LIN {X 0,Y 443.866,Z 651.881,A -85,B 0,C 180,E1 8636.588,E2 8636.588} C_VEL
LIN {X 0,Y 424.776,Z 822.719,A -85,B 0,C 180,E1 8634.304,E2 8634.304} C_VEL
LIN {X 0,Y 420.494,Z 848.982,A -85,B 0,C 180,E1 8633.917,E2 8633.917} C_VEL
LIN {X 0,Y 414.112,Z 876.582,A -85,B 0,C 180,E1 8633.45,E2 8633.45} C_VEL
LIN {X 0,Y 407.99,Z 898.031,A -85,B 0,C 180,E1 8632.991,E2 8632.991} C_VEL
LIN {X 0,Y 400.93,Z 919.109,A -85,B 0,C 180,E1 8632.437,E2 8632.437} C_VEL
LIN {X 0,Y 392.51,Z 940.895,A -85,B 0,C 180,E1 8631.745,E2 8631.745} C_VEL
LIN {X 0,Y 380.405,Z 967.798,A -85,B 0,C 180,E1 8630.683,E2 8630.683} C_VEL
LIN {X 0,Y 369.913,Z 988.144,A -85,B 0,C 180,E1 8629.696,E2 8629.696} C_VEL
LIN {X 0,Y 359.109,Z 1007.066,A -85,B 0,C 180,E1 8628.598,E2 8628.598} C_VEL
LIN {X 0,Y 347.933,Z 1024.879,A -85,B 0,C 180,E1 8627.384,E2 8627.384} C_VEL
LIN {X 0,Y 333.364,Z 1046.114,A -85,B 0,C 180,E1 8625.643,E2 8625.643} C_VEL
LIN {X 0,Y 317.605,Z 1066.602,A -85,B 0,C 180,E1 8623.54,E2 8623.54} C_VEL
LIN {X 0,Y 304.112,Z 1082.781,A -85,B 0,C 180,E1 8621.51,E2 8621.51} C_VEL
LIN {X 0,Y 290.809,Z 1097.657,A -85,B 0,C 180,E1 8619.258,E2 8619.258} C_VEL
LIN {X 0,Y 275.048,Z 1114.162,A -85,B 0,C 180,E1 8616.201,E2 8616.201} C_VEL
LIN {X 0,Y 258.412,Z 1130.204,A -85,B 0,C 180,E1 8612.381,E2 8612.381} C_VEL
LIN {X 0,Y 245.42,Z 1142.096,A -85,B 0,C 180,E1 8608.821,E2 8608.821} C_VEL
LIN {X 0,Y 233.402,Z 1152.698,A -85,B 0,C 180,E1 8604.906,E2 8604.906} C_VEL
LIN {X 0,Y 221.406,Z 1163.045,A -85,B 0,C 180,E1 8600.148,E2 8600.148} C_VEL
LIN {X 0,Y 207.773,Z 1174.693,A -85,B 0,C 180,E1 8593.105,E2 8593.105} C_VEL
LIN {X 0,Y 199.178,Z 1182.245,A -85,B 0,C 180,E1 8587.041,E2 8587.041} C_VEL
LIN {X 0,Y 192.825,Z 1188.259,A -85,B 0,C 180,E1 8580.887,E2 8580.887} C_VEL
LIN {X 0,Y 188.308,Z 1193.142,A -85,B 0,C 180,E1 8574.466,E2 8574.466} C_VEL
LIN {X 0,Y 185.354,Z 1197.256,A -85,B 0,C 180,E1 8567.259,E2 8567.259} C_VEL
LIN {X 0,Y 184.079,Z 1200.28,A -85,B 0,C 180,E1 8559.378,E2 8559.378} C_VEL
LIN {X 0,Y 183.917,Z 1201.596,A -85,B 0,C 180,E1 8553.116,E2 8553.116} C_VEL
LIN {X 0,Y 183.913,Z 1201.997,A -85,B 0,C 180,E1 8547.507,E2 8547.507} C_VEL
LIN {X 0,Y 184.046,Z 1201.547,A -85,B 0,C 180,E1 8541.251,E2 8541.251} C_VEL
LIN {X 0,Y 185.236,Z 1199.666,A -85,B 0,C 180,E1 8533.377,E2 8533.377} C_VEL
LIN {X 0,Y 188.179,Z 1196.649,A -85,B 0,C 180,E1 8526.054,E2 8526.054} C_VEL
LIN {X 0,Y 192.95,Z 1192.697,A -85,B 0,C 180,E1 8519.343,E2 8519.343} C_VEL
LIN {X 0,Y 199.602,Z 1187.731,A -85,B 0,C 180,E1 8513.05,E2 8513.05} C_VEL
LIN {X 0,Y 208.813,Z 1181.234,A -85,B 0,C 180,E1 8506.786,E2 8506.786} C_VEL
LIN {X 0,Y 222.772,Z 1171.555,A -85,B 0,C 180,E1 8499.871,E2 8499.871} C_VEL
LIN {X 0,Y 236.844,Z 1161.509,A -85,B 0,C 180,E1 8494.593,E2 8494.593} C_VEL
LIN {X 0,Y 249.883,Z 1151.926,A -85,B 0,C 180,E1 8490.652,E2 8490.652} C_VEL
LIN {X 0,Y 263.952,Z 1141.12,A -85,B 0,C 180,E1 8487.104,E2 8487.104} C_VEL
LIN {X 0,Y 281.997,Z 1126.496,A -85,B 0,C 180,E1 8483.319,E2 8483.319} C_VEL
LIN {X 0,Y 300.287,Z 1110.217,A -85,B 0,C 180,E1 8480.122,E2 8480.122} C_VEL
LIN {X 0,Y 315.189,Z 1095.995,A -85,B 0,C 180,E1 8477.885,E2 8477.885} C_VEL
LIN {X 0,Y 329.674,Z 1081.143,A -85,B 0,C 180,E1 8475.968,E2 8475.968} C_VEL
LIN {X 0,Y 345.392,Z 1063.722,A -85,B 0,C 180,E1 8474.123,E2 8474.123} C_VEL
LIN {X 0,Y 363.236,Z 1041.735,A -85,B 0,C 180,E1 8472.263,E2 8472.263} C_VEL
LIN {X 0,Y 376.376,Z 1023.816,A -85,B 0,C 180,E1 8471.027,E2 8471.027} C_VEL
LIN {X 0,Y 388.341,Z 1005.955,A -85,B 0,C 180,E1 8469.997,E2 8469.997} C_VEL
LIN {X 0,Y 399.945,Z 986.891,A -85,B 0,C 180,E1 8469.072,E2 8469.072} C_VEL
LIN {X 0,Y 413.071,Z 962.812,A -85,B 0,C 180,E1 8468.109,E2 8468.109} C_VEL
LIN {X 0,Y 424.404,Z 938.434,A -85,B 0,C 180,E1 8467.327,E2 8467.327} C_VEL
LIN {X 0,Y 432.962,Z 917.372,A -85,B 0,C 180,E1 8466.777,E2 8466.777} C_VEL
LIN {X 0,Y 440.366,Z 896.336,A -85,B 0,C 180,E1 8466.323,E2 8466.323} C_VEL
LIN {X 0,Y 447.583,Z 872.049,A -85,B 0,C 180,E1 8465.902,E2 8465.902} C_VEL
LIN {X 0,Y 454.093,Z 843.665,A -85,B 0,C 180,E1 8465.507,E2 8465.507} C_VEL
LIN {X 0,Y 457.997,Z 820.681,A -85,B 0,C 180,E1 8465.208,E2 8465.208} C_VEL
LIN {X 0,Y 475.341,Z 679.715,A -85,B 0,C 180,E1 8463.437,E2 8463.437} C_VEL
LIN {X 0,Y 475.301,Z 680.039,A -85,B 0,C 180,E1 8463.377,E2 8463.377} C_VEL
LIN {X 0,Y 457.777,Z 822.091,A -85,B 0,C 180,E1 8461.612,E2 8461.612} C_VEL
LIN {X 0,Y 452.981,Z 849.333,A -85,B 0,C 180,E1 8461.256,E2 8461.256} C_VEL
LIN {X 0,Y 446.328,Z 876.186,A -85,B 0,C 180,E1 8460.853,E2 8460.853} C_VEL
LIN {X 0,Y 439.95,Z 897.255,A -85,B 0,C 180,E1 8460.454,E2 8460.454} C_VEL
LIN {X 0,Y 432.487,Z 918.241,A -85,B 0,C 180,E1 8459.972,E2 8459.972} C_VEL
LIN {X 0,Y 423.465,Z 940.191,A -85,B 0,C 180,E1 8459.362,E2 8459.362} C_VEL
LIN {X 0,Y 410.642,Z 966.852,A -85,B 0,C 180,E1 8458.444,E2 8458.444} C_VEL
LIN {X 0,Y 399.788,Z 986.536,A -85,B 0,C 180,E1 8457.615,E2 8457.615} C_VEL
LIN {X 0,Y 388.59,Z 1004.872,A -85,B 0,C 180,E1 8456.696,E2 8456.696} C_VEL
LIN {X 0,Y 376.533,Z 1022.797,A -85,B 0,C 180,E1 8455.644,E2 8455.644} C_VEL
LIN {X 0,Y 362.532,Z 1041.768,A -85,B 0,C 180,E1 8454.302,E2 8454.302} C_VEL
LIN {X 0,Y 344.561,Z 1063.586,A -85,B 0,C 180,E1 8452.39,E2 8452.39} C_VEL
LIN {X 0,Y 330.011,Z 1079.597,A -85,B 0,C 180,E1 8450.651,E2 8450.651} C_VEL
LIN {X 0,Y 315.549,Z 1094.316,A -85,B 0,C 180,E1 8448.721,E2 8448.721} C_VEL
LIN {X 0,Y 300.35,Z 1108.691,A -85,B 0,C 180,E1 8446.424,E2 8446.424} C_VEL
LIN {X 0,Y 281.29,Z 1125.37,A -85,B 0,C 180,E1 8443.053,E2 8443.053} C_VEL
LIN {X 0,Y 264.66,Z 1138.691,A -85,B 0,C 180,E1 8439.54,E2 8439.54} C_VEL
LIN {X 0,Y 250.503,Z 1149.41,A -85,B 0,C 180,E1 8435.975,E2 8435.975} C_VEL
LIN {X 0,Y 236.953,Z 1159.197,A -85,B 0,C 180,E1 8431.873,E2 8431.873} C_VEL
LIN {X 0,Y 221.703,Z 1169.857,A -85,B 0,C 180,E1 8426.08,E2 8426.08} C_VEL
LIN {X 0,Y 208.814,Z 1178.482,A -85,B 0,C 180,E1 8419.582,E2 8419.582} C_VEL
LIN {X 0,Y 199.873,Z 1184.582,A -85,B 0,C 180,E1 8413.499,E2 8413.499} C_VEL
LIN {X 0,Y 193.099,Z 1189.424,A -85,B 0,C 180,E1 8407.114,E2 8407.114} C_VEL
LIN {X 0,Y 187.925,Z 1193.548,A -85,B 0,C 180,E1 8399.657,E2 8399.657} C_VEL
LIN {X 0,Y 184.898,Z 1196.483,A -85,B 0,C 180,E1 8391.242,E2 8391.242} C_VEL
LIN {X 0,Y 184.057,Z 1197.676,A -85,B 0,C 180,E1 8384.471,E2 8384.471} C_VEL
LIN {X 0,Y 183.922,Z 1197.904,A -85,B 0,C 180,E1 8378.331,E2 8378.331} C_VEL
LIN {X 0,Y 183.937,Z 1197.343,A -85,B 0,C 180,E1 8372.492,E2 8372.492} C_VEL
LIN {X 0,Y 184.312,Z 1195.758,A -85,B 0,C 180,E1 8365.956,E2 8365.956} C_VEL
LIN {X 0,Y 185.733,Z 1193.043,A -85,B 0,C 180,E1 8359.14,E2 8359.14} C_VEL
LIN {X 0,Y 188.713,Z 1189.247,A -85,B 0,C 180,E1 8352.422,E2 8352.422} C_VEL
LIN {X 0,Y 193.222,Z 1184.592,A -85,B 0,C 180,E1 8346.195,E2 8346.195} C_VEL
LIN {X 0,Y 199.432,Z 1178.892,A -85,B 0,C 180,E1 8340.242,E2 8340.242} C_VEL
LIN {X 0,Y 207.741,Z 1171.761,A -85,B 0,C 180,E1 8334.383,E2 8334.383} C_VEL
LIN {X 0,Y 219.756,Z 1161.785,A -85,B 0,C 180,E1 8328.024,E2 8328.024} C_VEL
LIN {X 0,Y 233.341,Z 1150.204,A -85,B 0,C 180,E1 8322.523,E2 8322.523} C_VEL
LIN {X 0,Y 245.468,Z 1139.649,A -85,B 0,C 180,E1 8318.55,E2 8318.55} C_VEL
LIN {X 0,Y 258.583,Z 1127.787,A -85,B 0,C 180,E1 8314.942,E2 8314.942} C_VEL
LIN {X 0,Y 274.719,Z 1112.442,A -85,B 0,C 180,E1 8311.208,E2 8311.208} C_VEL
LIN {X 0,Y 291.052,Z 1095.466,A -85,B 0,C 180,E1 8308.009,E2 8308.009} C_VEL
LIN {X 0,Y 304.218,Z 1080.858,A -85,B 0,C 180,E1 8305.771,E2 8305.771} C_VEL
LIN {X 0,Y 317.272,Z 1065.327,A -85,B 0,C 180,E1 8303.791,E2 8303.791} C_VEL
LIN {X 0,Y 330.9,Z 1047.812,A -85,B 0,C 180,E1 8301.931,E2 8301.931} C_VEL
LIN {X 0,Y 346.823,Z 1025.164,A -85,B 0,C 180,E1 8299.978,E2 8299.978} C_VEL
LIN {X 0,Y 358.772,Z 1006.257,A -85,B 0,C 180,E1 8298.641,E2 8298.641} C_VEL
LIN {X 0,Y 369.602,Z 987.426,A -85,B 0,C 180,E1 8297.524,E2 8297.524} C_VEL
LIN {X 0,Y 379.674,Z 968.031,A -85,B 0,C 180,E1 8296.549,E2 8296.549} C_VEL
LIN {X 0,Y 391.196,Z 943.066,A -85,B 0,C 180,E1 8295.513,E2 8295.513} C_VEL
LIN {X 0,Y 400.78,Z 918.46,A -85,B 0,C 180,E1 8294.691,E2 8294.691} C_VEL
LIN {X 0,Y 407.769,Z 897.72,A -85,B 0,C 180,E1 8294.124,E2 8294.124} C_VEL
LIN {X 0,Y 413.868,Z 876.495,A -85,B 0,C 180,E1 8293.643,E2 8293.643} C_VEL
LIN {X 0,Y 419.539,Z 852.593,A -85,B 0,C 180,E1 8293.209,E2 8293.209} C_VEL
LIN {X 0,Y 424.62,Z 823.336,A -85,B 0,C 180,E1 8292.774,E2 8292.774} C_VEL
LIN {X 0,Y 432.472,Z 754.37,A -85,B 0,C 180,E1 8291.843,E2 8291.843} C_VEL
LIN {X 0,Y 443.846,Z 651.537,A -85,B 0,C 180,E1 8290.448,E2 8290.448} C_VEL
LIN {X 0,Y 442.904,Z 649.337,A -85,B 0,C 180,E1 8288.962,E2 8288.962} C_VEL
LIN {X 0,Y 441.948,Z 646.598,A -85,B 0,C 180,E1 8286.693,E2 8286.693} C_VEL
LIN {X 0,Y 441.415,Z 645.936,A -85,B 0,C 180,E1 8282.857,E2 8282.857} C_VEL
LIN {X 0,Y 441.662,Z 646.287,A -85,B 0,C 180,E1 8281.327,E2 8281.327} C_VEL
LIN {X 0,Y 441.718,Z 647.33,A -85,B 0,C 180,E1 8280.766,E2 8280.766} C_VEL
LIN {X 0,Y 441.574,Z 651.709,A -85,B 0,C 180,E1 8279.845,E2 8279.845} C_VEL
LIN {X 0,Y 441.535,Z 655.781,A -85,B 0,C 180,E1 8279.002,E2 8279.002} C_VEL
LIN {X 0,Y 441.696,Z 656.897,A -85,B 0,C 180,E1 8278.534,E2 8278.534} C_VEL
LIN {X 0,Y 442.275,Z 658.15,A -85,B 0,C 180,E1 8277.538,E2 8277.538} C_VEL
LIN {X 0,Y 423.591,Z 822.639,A -85,B 0,C 180,E1 8275.377,E2 8275.377} C_VEL
LIN {X 0,Y 419.223,Z 849.082,A -85,B 0,C 180,E1 8274.997,E2 8274.997} C_VEL
LIN {X 0,Y 412.777,Z 876.62,A -85,B 0,C 180,E1 8274.547,E2 8274.547} C_VEL
LIN {X 0,Y 406.591,Z 898.047,A -85,B 0,C 180,E1 8274.105,E2 8274.105} C_VEL
LIN {X 0,Y 399.454,Z 919.109,A -85,B 0,C 180,E1 8273.571,E2 8273.571} C_VEL
LIN {X 0,Y 390.939,Z 940.883,A -85,B 0,C 180,E1 8272.903,E2 8272.903} C_VEL
LIN {X 0,Y 378.497,Z 968.138,A -85,B 0,C 180,E1 8271.862,E2 8271.862} C_VEL
LIN {X 0,Y 367.593,Z 988.937,A -85,B 0,C 180,E1 8270.881,E2 8270.881} C_VEL
LIN {X 0,Y 356.811,Z 1007.503,A -85,B 0,C 180,E1 8269.831,E2 8269.831} C_VEL
LIN {X 0,Y 344.78,Z 1026.326,A -85,B 0,C 180,E1 8268.577,E2 8268.577} C_VEL
LIN {X 0,Y 328.296,Z 1049.535,A -85,B 0,C 180,E1 8266.672,E2 8266.672} C_VEL
LIN {X 0,Y 313.919,Z 1067.729,A -85,B 0,C 180,E1 8264.813,E2 8264.813} C_VEL
LIN {X 0,Y 300.669,Z 1083.249,A -85,B 0,C 180,E1 8262.893,E2 8262.893} C_VEL
LIN {X 0,Y 286.303,Z 1098.905,A -85,B 0,C 180,E1 8260.547,E2 8260.547} C_VEL
LIN {X 0,Y 268.106,Z 1117.205,A -85,B 0,C 180,E1 8257.094,E2 8257.094} C_VEL
LIN {X 0,Y 253.141,Z 1131.12,A -85,B 0,C 180,E1 8253.715,E2 8253.715} C_VEL
LIN {X 0,Y 239.782,Z 1142.917,A -85,B 0,C 180,E1 8250.15,E2 8250.15} C_VEL
LIN {X 0,Y 226.515,Z 1154.166,A -85,B 0,C 180,E1 8245.902,E2 8245.902} C_VEL
LIN {X 0,Y 211.151,Z 1166.776,A -85,B 0,C 180,E1 8239.674,E2 8239.674} C_VEL
LIN {X 0,Y 200.341,Z 1175.532,A -85,B 0,C 180,E1 8233.925,E2 8233.925} C_VEL
LIN {X 0,Y 191.817,Z 1182.641,A -85,B 0,C 180,E1 8227.958,E2 8227.958} C_VEL
LIN {X 0,Y 185.167,Z 1188.578,A -85,B 0,C 180,E1 8221.586,E2 8221.586} C_VEL
LIN {X 0,Y 180.081,Z 1193.81,A -85,B 0,C 180,E1 8214.259,E2 8214.259} C_VEL
LIN {X 0,Y 176.939,Z 1198.115,A -85,B 0,C 180,E1 8205.738,E2 8205.738} C_VEL
LIN {X 0,Y 176.03,Z 1200.441,A -85,B 0,C 180,E1 8198.492,E2 8198.492} C_VEL
LIN {X 0,Y 175.917,Z 1201.568,A -85,B 0,C 180,E1 8192.28,E2 8192.28} C_VEL
LIN {X 0,Y 175.914,Z 1201.879,A -85,B 0,C 180,E1 8186.415,E2 8186.415} C_VEL
LIN {X 0,Y 176.136,Z 1201.318,A -85,B 0,C 180,E1 8179.865,E2 8179.865} C_VEL
LIN {X 0,Y 177.612,Z 1199.394,A -85,B 0,C 180,E1 8171.964,E2 8171.964} C_VEL
LIN {X 0,Y 180.976,Z 1196.369,A -85,B 0,C 180,E1 8164.473,E2 8164.473} C_VEL
LIN {X 0,Y 186.011,Z 1192.573,A -85,B 0,C 180,E1 8157.849,E2 8157.849} C_VEL
LIN {X 0,Y 193.206,Z 1187.609,A -85,B 0,C 180,E1 8151.395,E2 8151.395} C_VEL
LIN {X 0,Y 202.782,Z 1181.279,A -85,B 0,C 180,E1 8145.163,E2 8145.163} C_VEL
LIN {X 0,Y 217.489,Z 1171.647,A -85,B 0,C 180,E1 8138.175,E2 8138.175} C_VEL
LIN {X 0,Y 232.357,Z 1161.509,A -85,B 0,C 180,E1 8132.834,E2 8132.834} C_VEL
LIN {X 0,Y 246.427,Z 1151.562,A -85,B 0,C 180,E1 8128.789,E2 8128.789} C_VEL
LIN {X 0,Y 262.191,Z 1139.838,A -85,B 0,C 180,E1 8125.044,E2 8125.044} C_VEL
LIN {X 0,Y 282.812,Z 1123.293,A -85,B 0,C 180,E1 8121.037,E2 8121.037} C_VEL
LIN {X 0,Y 298.379,Z 1109.731,A -85,B 0,C 180,E1 8118.5,E2 8118.5} C_VEL
LIN {X 0,Y 313.615,Z 1095.474,A -85,B 0,C 180,E1 8116.334,E2 8116.334} C_VEL
LIN {X 0,Y 329.267,Z 1079.67,A -85,B 0,C 180,E1 8114.378,E2 8114.378} C_VEL
LIN {X 0,Y 347.977,Z 1058.932,A -85,B 0,C 180,E1 8112.33,E2 8112.33} C_VEL
LIN {X 0,Y 363.426,Z 1039.824,A -85,B 0,C 180,E1 8110.834,E2 8110.834} C_VEL
LIN {X 0,Y 375.647,Z 1023.311,A -85,B 0,C 180,E1 8109.754,E2 8109.754} C_VEL
LIN {X 0,Y 388.023,Z 1005.022,A -85,B 0,C 180,E1 8108.745,E2 8108.745} C_VEL
LIN {X 0,Y 400.176,Z 985.189,A -85,B 0,C 180,E1 8107.832,E2 8107.832} C_VEL
LIN {X 0,Y 414.396,Z 958.757,A -85,B 0,C 180,E1 8106.848,E2 8106.848} C_VEL
LIN {X 0,Y 424.422,Z 937.2,A -85,B 0,C 180,E1 8106.201,E2 8106.201} C_VEL
LIN {X 0,Y 432.608,Z 917.166,A -85,B 0,C 180,E1 8105.704,E2 8105.704} C_VEL
LIN {X 0,Y 440.048,Z 896.191,A -85,B 0,C 180,E1 8105.272,E2 8105.272} C_VEL
LIN {X 0,Y 447.445,Z 871.471,A -85,B 0,C 180,E1 8104.864,E2 8104.864} C_VEL
LIN {X 0,Y 453.921,Z 843.316,A -85,B 0,C 180,E1 8104.489,E2 8104.489} C_VEL
LIN {X 0,Y 457.835,Z 820.461,A -85,B 0,C 180,E1 8104.2,E2 8104.2} C_VEL
LIN {X 0,Y 465.839,Z 756.902,A -85,B 0,C 180,E1 8103.416,E2 8103.416} C_VEL
LIN {X 0,Y 457.308,Z 824.05,A -85,B 0,C 180,E1 8102.593,E2 8102.593} C_VEL
LIN {X 0,Y 451.773,Z 853.513,A -85,B 0,C 180,E1 8102.217,E2 8102.217} C_VEL
LIN {X 0,Y 445.735,Z 877.298,A -85,B 0,C 180,E1 8101.868,E2 8101.868} C_VEL
LIN {X 0,Y 439.334,Z 898.118,A -85,B 0,C 180,E1 8101.487,E2 8101.487} C_VEL
LIN {X 0,Y 431.756,Z 919.132,A -85,B 0,C 180,E1 8101.022,E2 8101.022} C_VEL
LIN {X 0,Y 421.447,Z 943.771,A -85,B 0,C 180,E1 8100.355,E2 8100.355} C_VEL
LIN {X 0,Y 409.454,Z 967.959,A -85,B 0,C 180,E1 8099.539,E2 8099.539} C_VEL
LIN {X 0,Y 398.416,Z 987.662,A -85,B 0,C 180,E1 8098.737,E2 8098.737} C_VEL
LIN {X 0,Y 387.213,Z 1005.699,A -85,B 0,C 180,E1 8097.862,E2 8097.862} C_VEL
LIN {X 0,Y 374.286,Z 1024.573,A -85,B 0,C 180,E1 8096.784,E2 8096.784} C_VEL
LIN {X 0,Y 357.199,Z 1047.006,A -85,B 0,C 180,E1 8095.205,E2 8095.205} C_VEL
LIN {X 0,Y 341.112,Z 1065.81,A -85,B 0,C 180,E1 8093.547,E2 8093.547} C_VEL
LIN {X 0,Y 326.901,Z 1081.067,A -85,B 0,C 180,E1 8091.912,E2 8091.912} C_VEL
LIN {X 0,Y 312.319,Z 1095.543,A -85,B 0,C 180,E1 8090.045,E2 8090.045} C_VEL
LIN {X 0,Y 294.087,Z 1112.307,A -85,B 0,C 180,E1 8087.359,E2 8087.359} C_VEL
LIN {X 0,Y 275.458,Z 1127.784,A -85,B 0,C 180,E1 8084.132,E2 8084.132} C_VEL
LIN {X 0,Y 260.158,Z 1139.635,A -85,B 0,C 180,E1 8080.987,E2 8080.987} C_VEL
LIN {X 0,Y 245.71,Z 1150.175,A -85,B 0,C 180,E1 8077.476,E2 8077.476} C_VEL
LIN {X 0,Y 230.097,Z 1161.006,A -85,B 0,C 180,E1 8072.853,E2 8072.853} C_VEL
LIN {X 0,Y 213.993,Z 1171.545,A -85,B 0,C 180,E1 8066.757,E2 8066.757} C_VEL
LIN {X 0,Y 202.271,Z 1179.018,A -85,B 0,C 180,E1 8060.902,E2 8060.902} C_VEL
LIN {X 0,Y 193.019,Z 1184.94,A -85,B 0,C 180,E1 8054.788,E2 8054.788} C_VEL
LIN {X 0,Y 185.538,Z 1189.926,A -85,B 0,C 180,E1 8047.904,E2 8047.904} C_VEL
LIN {X 0,Y 179.5,Z 1194.401,A -85,B 0,C 180,E1 8038.987,E2 8038.987} C_VEL
LIN {X 0,Y 176.855,Z 1196.755,A -85,B 0,C 180,E1 8031.113,E2 8031.113} C_VEL
LIN {X 0,Y 176.057,Z 1197.796,A -85,B 0,C 180,E1 8024.471,E2 8024.471} C_VEL
LIN {X 0,Y 175.925,Z 1197.989,A -85,B 0,C 180,E1 8018.498,E2 8018.498} C_VEL
LIN {X 0,Y 175.935,Z 1197.468,A -85,B 0,C 180,E1 8012.606,E2 8012.606} C_VEL
LIN {X 0,Y 176.329,Z 1195.908,A -85,B 0,C 180,E1 8005.773,E2 8005.773} C_VEL
LIN {X 0,Y 177.957,Z 1193.062,A -85,B 0,C 180,E1 7998.331,E2 7998.331} C_VEL
LIN {X 0,Y 181.232,Z 1189.246,A -85,B 0,C 180,E1 7991.338,E2 7991.338} C_VEL
LIN {X 0,Y 186.119,Z 1184.571,A -85,B 0,C 180,E1 7984.887,E2 7984.887} C_VEL
LIN {X 0,Y 193.152,Z 1178.554,A -85,B 0,C 180,E1 7978.478,E2 7978.478} C_VEL
LIN {X 0,Y 202.972,Z 1170.664,A -85,B 0,C 180,E1 7971.993,E2 7971.993} C_VEL
LIN {X 0,Y 216.842,Z 1159.569,A -85,B 0,C 180,E1 7965.245,E2 7965.245} C_VEL
LIN {X 0,Y 229.431,Z 1149.313,A -85,B 0,C 180,E1 7960.494,E2 7960.494} C_VEL
LIN {X 0,Y 242.458,Z 1138.367,A -85,B 0,C 180,E1 7956.472,E2 7956.472} C_VEL
LIN {X 0,Y 258.969,Z 1123.858,A -85,B 0,C 180,E1 7952.271,E2 7952.271} C_VEL
LIN {X 0,Y 275.099,Z 1108.429,A -85,B 0,C 180,E1 7948.846,E2 7948.846} C_VEL
LIN {X 0,Y 288.91,Z 1094.347,A -85,B 0,C 180,E1 7946.319,E2 7946.319} C_VEL
LIN {X 0,Y 302.407,Z 1079.62,A -85,B 0,C 180,E1 7944.141,E2 7944.141} C_VEL
LIN {X 0,Y 317.118,Z 1062.327,A -85,B 0,C 180,E1 7942.034,E2 7942.034} C_VEL
LIN {X 0,Y 333.898,Z 1040.514,A -85,B 0,C 180,E1 7939.903,E2 7939.903} C_VEL
LIN {X 0,Y 346.756,Z 1022.021,A -85,B 0,C 180,E1 7938.44,E2 7938.44} C_VEL
LIN {X 0,Y 358.055,Z 1004.214,A -85,B 0,C 180,E1 7937.25,E2 7937.25} C_VEL
LIN {X 0,Y 369.494,Z 984.356,A -85,B 0,C 180,E1 7936.13,E2 7936.13} C_VEL
LIN {X 0,Y 382.413,Z 959.013,A -85,B 0,C 180,E1 7934.963,E2 7934.963} C_VEL
LIN {X 0,Y 392.303,Z 936.538,A -85,B 0,C 180,E1 7934.124,E2 7934.124} C_VEL
LIN {X 0,Y 400.001,Z 916.643,A -85,B 0,C 180,E1 7933.503,E2 7933.503} C_VEL
LIN {X 0,Y 407.058,Z 895.657,A -85,B 0,C 180,E1 7932.958,E2 7932.958} C_VEL
LIN {X 0,Y 413.773,Z 872.042,A -85,B 0,C 180,E1 7932.455,E2 7932.455} C_VEL
LIN {X 0,Y 420.13,Z 843.287,A -85,B 0,C 180,E1 7931.986,E2 7931.986} C_VEL
LIN {X 0,Y 423.868,Z 820.064,A -85,B 0,C 180,E1 7931.656,E2 7931.656} C_VEL
LIN {X 0,Y 442.263,Z 658.004,A -85,B 0,C 180,E1 7929.529,E2 7929.529} C_VEL
LIN {X 0,Y 440.949,Z 654.526,A -85,B 0,C 180,E1 7926.641,E2 7926.641} C_VEL
LIN {X 0,Y 440.437,Z 653.878,A -85,B 0,C 180,E1 7922.863,E2 7922.863} C_VEL
LIN {X 0,Y 441.06,Z 654.792,A -85,B 0,C 180,E1 7920.13,E2 7920.13} C_VEL
LIN {X 0,Y 441.696,Z 656.897,A -85,B 0,C 180,E1 7918.534,E2 7918.534} C_VEL
LIN {X 0,Y 441.712,Z 658.232,A -85,B 0,C 180,E1 7918.27,E2 7918.27} C_VEL
LIN {X 0,Y 441.466,Z 661.243,A -85,B 0,C 180,E1 7918.094,E2 7918.094} C_VEL
LIN {X 0,Y 440.865,Z 666.276,A -85,B 0,C 180,E1 7918.065,E2 7918.065} C_VEL
LIN {X 0,Y 439.256,Z 677.952,A -85,B 0,C 180,E1 7918.297,E2 7918.297} C_VEL
LIN {X 0,Y 438.927,Z 680.662,A -85,B 0,C 180,E1 7918.288,E2 7918.288} C_VEL
LIN {X 0,Y 422.55,Z 822.596,A -85,B 0,C 180,E1 7916.456,E2 7916.456} C_VEL
LIN {X 0,Y 418.103,Z 849.182,A -85,B 0,C 180,E1 7916.084,E2 7916.084} C_VEL
LIN {X 0,Y 411.594,Z 876.657,A -85,B 0,C 180,E1 7915.65,E2 7915.65} C_VEL
LIN {X 0,Y 405.347,Z 898.064,A -85,B 0,C 180,E1 7915.226,E2 7915.226} C_VEL
LIN {X 0,Y 398.309,Z 918.638,A -85,B 0,C 180,E1 7914.725,E2 7914.725} C_VEL
LIN {X 0,Y 390.004,Z 939.714,A -85,B 0,C 180,E1 7914.107,E2 7914.107} C_VEL
LIN {X 0,Y 378.143,Z 965.765,A -85,B 0,C 180,E1 7913.166,E2 7913.166} C_VEL
LIN {X 0,Y 366.369,Z 988.068,A -85,B 0,C 180,E1 7912.163,E2 7912.163} C_VEL
LIN {X 0,Y 355.715,Z 1006.254,A -85,B 0,C 180,E1 7911.179,E2 7911.179} C_VEL
LIN {X 0,Y 344.136,Z 1024.221,A -85,B 0,C 180,E1 7910.041,E2 7910.041} C_VEL
LIN {X 0,Y 330.058,Z 1044.154,A -85,B 0,C 180,E1 7908.518,E2 7908.518} C_VEL
LIN {X 0,Y 313.143,Z 1065.6,A -85,B 0,C 180,E1 7906.472,E2 7906.472} C_VEL
LIN {X 0,Y 298.811,Z 1082.158,A -85,B 0,C 180,E1 7904.51,E2 7904.51} C_VEL
LIN {X 0,Y 285.275,Z 1096.68,A -85,B 0,C 180,E1 7902.426,E2 7902.426} C_VEL
LIN {X 0,Y 270.948,Z 1111.019,A -85,B 0,C 180,E1 7899.928,E2 7899.928} C_VEL
LIN {X 0,Y 252.81,Z 1127.892,A -85,B 0,C 180,E1 7896.208,E2 7896.208} C_VEL
LIN {X 0,Y 237.104,Z 1141.381,A -85,B 0,C 180,E1 7892.32,E2 7892.32} C_VEL
LIN {X 0,Y 224.102,Z 1152.041,A -85,B 0,C 180,E1 7888.448,E2 7888.448} C_VEL
LIN {X 0,Y 211.554,Z 1161.968,A -85,B 0,C 180,E1 7883.919,E2 7883.919} C_VEL
LIN {X 0,Y 197.804,Z 1172.733,A -85,B 0,C 180,E1 7877.561,E2 7877.561} C_VEL
LIN {X 0,Y 186.342,Z 1181.575,A -85,B 0,C 180,E1 7870.363,E2 7870.363} C_VEL
LIN {X 0,Y 179.025,Z 1187.591,A -85,B 0,C 180,E1 7863.952,E2 7863.952} C_VEL
LIN {X 0,Y 173.59,Z 1192.569,A -85,B 0,C 180,E1 7857.067,E2 7857.067} C_VEL
LIN {X 0,Y 170.113,Z 1196.449,A -85,B 0,C 180,E1 7849.932,E2 7849.932} C_VEL
LIN {X 0,Y 168.431,Z 1199.141,A -85,B 0,C 180,E1 7843.037,E2 7843.037} C_VEL
LIN {X 0,Y 167.965,Z 1200.741,A -85,B 0,C 180,E1 7836.837,E2 7836.837} C_VEL
LIN {X 0,Y 167.921,Z 1201.538,A -85,B 0,C 180,E1 7831.365,E2 7831.365} C_VEL
LIN {X 0,Y 167.918,Z 1201.753,A -85,B 0,C 180,E1 7825.56,E2 7825.56} C_VEL
LIN {X 0,Y 168.243,Z 1201.119,A -85,B 0,C 180,E1 7818.69,E2 7818.69} C_VEL
LIN {X 0,Y 169.955,Z 1199.239,A -85,B 0,C 180,E1 7810.765,E2 7810.765} C_VEL
LIN {X 0,Y 173.609,Z 1196.309,A -85,B 0,C 180,E1 7803.217,E2 7803.217} C_VEL
LIN {X 0,Y 179.334,Z 1192.366,A -85,B 0,C 180,E1 7796.114,E2 7796.114} C_VEL
LIN {X 0,Y 187.335,Z 1187.269,A -85,B 0,C 180,E1 7789.372,E2 7789.372} C_VEL
LIN {X 0,Y 199.14,Z 1180.013,A -85,B 0,C 180,E1 7782.285,E2 7782.285} C_VEL
LIN {X 0,Y 214.822,Z 1170.137,A -85,B 0,C 180,E1 7775.461,E2 7775.461} C_VEL
LIN {X 0,Y 228.423,Z 1161.294,A -85,B 0,C 180,E1 7770.915,E2 7770.915} C_VEL
LIN {X 0,Y 242.511,Z 1151.711,A -85,B 0,C 180,E1 7767.057,E2 7767.057} C_VEL
LIN {X 0,Y 258.02,Z 1140.562,A -85,B 0,C 180,E1 7763.525,E2 7763.525} C_VEL
LIN {X 0,Y 277.477,Z 1125.604,A -85,B 0,C 180,E1 7759.868,E2 7759.868} C_VEL
LIN {X 0,Y 295.861,Z 1110.007,A -85,B 0,C 180,E1 7756.983,E2 7756.983} C_VEL
LIN {X 0,Y 311.399,Z 1095.784,A -85,B 0,C 180,E1 7754.88,E2 7754.88} C_VEL
LIN {X 0,Y 326.432,Z 1080.928,A -85,B 0,C 180,E1 7753.087,E2 7753.087} C_VEL
LIN {X 0,Y 343.592,Z 1062.503,A -85,B 0,C 180,E1 7751.283,E2 7751.283} C_VEL
LIN {X 0,Y 361.062,Z 1041.505,A -85,B 0,C 180,E1 7749.654,E2 7749.654} C_VEL
LIN {X 0,Y 374.579,Z 1023.563,A -85,B 0,C 180,E1 7748.519,E2 7748.519} C_VEL
LIN {X 0,Y 387.29,Z 1005.015,A -85,B 0,C 180,E1 7747.537,E2 7747.537} C_VEL
LIN {X 0,Y 399.64,Z 985.078,A -85,B 0,C 180,E1 7746.661,E2 7746.661} C_VEL
LIN {X 0,Y 414.002,Z 958.638,A -85,B 0,C 180,E1 7745.72,E2 7745.72} C_VEL
LIN {X 0,Y 424.129,Z 937.054,A -85,B 0,C 180,E1 7745.104,E2 7745.104} C_VEL
LIN {X 0,Y 432.35,Z 917.103,A -85,B 0,C 180,E1 7744.633,E2 7744.633} C_VEL
LIN {X 0,Y 439.636,Z 896.772,A -85,B 0,C 180,E1 7744.233,E2 7744.233} C_VEL
LIN {X 0,Y 446.579,Z 873.946,A -85,B 0,C 180,E1 7743.87,E2 7743.87} C_VEL
LIN {X 0,Y 453.649,Z 844.231,A -85,B 0,C 180,E1 7743.486,E2 7743.486} C_VEL
LIN {X 0,Y 454.632,Z 839.124,A -85,B 0,C 180,E1 7743.417,E2 7743.417} C_VEL
LIN {X 0,Y 449.814,Z 861.311,A -85,B 0,C 180,E1 7743.136,E2 7743.136} C_VEL
LIN {X 0,Y 443.17,Z 885.764,A -85,B 0,C 180,E1 7742.764,E2 7742.764} C_VEL
LIN {X 0,Y 433.816,Z 913.165,A -85,B 0,C 180,E1 7742.231,E2 7742.231} C_VEL
LIN {X 0,Y 425.128,Z 934.575,A -85,B 0,C 180,E1 7741.714,E2 7741.714} C_VEL
LIN {X 0,Y 416.022,Z 954.253,A -85,B 0,C 180,E1 7741.141,E2 7741.141} C_VEL
LIN {X 0,Y 405.585,Z 974.271,A -85,B 0,C 180,E1 7740.449,E2 7740.449} C_VEL
LIN {X 0,Y 391.461,Z 998.248,A -85,B 0,C 180,E1 7739.444,E2 7739.444} C_VEL
LIN {X 0,Y 376.954,Z 1019.723,A -85,B 0,C 180,E1 7738.328,E2 7738.328} C_VEL
LIN {X 0,Y 363.737,Z 1037.446,A -85,B 0,C 180,E1 7737.21,E2 7737.21} C_VEL
LIN {X 0,Y 350.31,Z 1053.905,A -85,B 0,C 180,E1 7735.982,E2 7735.982} C_VEL
LIN {X 0,Y 334.091,Z 1072.108,A -85,B 0,C 180,E1 7734.332,E2 7734.332} C_VEL
LIN {X 0,Y 314.931,Z 1091.418,A -85,B 0,C 180,E1 7732.117,E2 7732.117} C_VEL
LIN {X 0,Y 298.55,Z 1106.454,A -85,B 0,C 180,E1 7729.937,E2 7729.937} C_VEL
LIN {X 0,Y 283.52,Z 1119.24,A -85,B 0,C 180,E1 7727.65,E2 7727.65} C_VEL
LIN {X 0,Y 267.312,Z 1132.073,A -85,B 0,C 180,E1 7724.802,E2 7724.802} C_VEL
LIN {X 0,Y 247.117,Z 1146.823,A -85,B 0,C 180,E1 7720.517,E2 7720.517} C_VEL
LIN {X 0,Y 230.897,Z 1157.749,A -85,B 0,C 180,E1 7716.251,E2 7716.251} C_VEL
LIN {X 0,Y 217.546,Z 1166.301,A -85,B 0,C 180,E1 7711.938,E2 7711.938} C_VEL
LIN {X 0,Y 204.566,Z 1174.313,A -85,B 0,C 180,E1 7706.699,E2 7706.699} C_VEL
LIN {X 0,Y 190.491,Z 1182.827,A -85,B 0,C 180,E1 7699.098,E2 7699.098} C_VEL
LIN {X 0,Y 180.784,Z 1188.65,A -85,B 0,C 180,E1 7691.581,E2 7691.581} C_VEL
LIN {X 0,Y 174.626,Z 1192.588,A -85,B 0,C 180,E1 7684.53,E2 7684.53} C_VEL
LIN {X 0,Y 170.79,Z 1195.334,A -85,B 0,C 180,E1 7677.548,E2 7677.548} C_VEL
LIN {X 0,Y 168.733,Z 1197.106,A -85,B 0,C 180,E1 7670.562,E2 7670.562} C_VEL
LIN {X 0,Y 168.056,Z 1197.916,A -85,B 0,C 180,E1 7664.47,E2 7664.47} C_VEL
LIN {X 0,Y 167.925,Z 1198.067,A -85,B 0,C 180,E1 7658.561,E2 7658.561} C_VEL
LIN {X 0,Y 167.939,Z 1197.525,A -85,B 0,C 180,E1 7652.389,E2 7652.389} C_VEL
LIN {X 0,Y 168.348,Z 1196.057,A -85,B 0,C 180,E1 7645.572,E2 7645.572} C_VEL
LIN {X 0,Y 170.097,Z 1193.237,A -85,B 0,C 180,E1 7637.783,E2 7637.783} C_VEL
LIN {X 0,Y 173.611,Z 1189.447,A -85,B 0,C 180,E1 7630.486,E2 7630.486} C_VEL
LIN {X 0,Y 178.826,Z 1184.799,A -85,B 0,C 180,E1 7623.787,E2 7623.787} C_VEL
LIN {X 0,Y 185.904,Z 1179.104,A -85,B 0,C 180,E1 7617.464,E2 7617.464} C_VEL
LIN {X 0,Y 195.222,Z 1171.978,A -85,B 0,C 180,E1 7611.33,E2 7611.33} C_VEL
LIN {X 0,Y 208.516,Z 1162.01,A -85,B 0,C 180,E1 7604.792,E2 7604.792} C_VEL
LIN {X 0,Y 223.291,Z 1150.435,A -85,B 0,C 180,E1 7599.226,E2 7599.226} C_VEL
LIN {X 0,Y 236.357,Z 1139.882,A -85,B 0,C 180,E1 7595.27,E2 7595.27} C_VEL
LIN {X 0,Y 249.637,Z 1128.642,A -85,B 0,C 180,E1 7591.885,E2 7591.885} C_VEL
LIN {X 0,Y 265.159,Z 1114.737,A -85,B 0,C 180,E1 7588.527,E2 7588.527} C_VEL
LIN {X 0,Y 283.029,Z 1097.358,A -85,B 0,C 180,E1 7585.262,E2 7585.262} C_VEL
LIN {X 0,Y 298.027,Z 1081.484,A -85,B 0,C 180,E1 7582.904,E2 7582.904} C_VEL
LIN {X 0,Y 311.667,Z 1065.915,A -85,B 0,C 180,E1 7581.005,E2 7581.005} C_VEL
LIN {X 0,Y 325.246,Z 1049.136,A -85,B 0,C 180,E1 7579.307,E2 7579.307} C_VEL
LIN {X 0,Y 341.691,Z 1026.704,A -85,B 0,C 180,E1 7577.458,E2 7577.458} C_VEL
LIN {X 0,Y 354.884,Z 1006.48,A -85,B 0,C 180,E1 7576.109,E2 7576.109} C_VEL
LIN {X 0,Y 366.063,Z 987.564,A -85,B 0,C 180,E1 7575.055,E2 7575.055} C_VEL
LIN {X 0,Y 376.397,Z 968.181,A -85,B 0,C 180,E1 7574.146,E2 7574.146} C_VEL
LIN {X 0,Y 388.172,Z 943.287,A -85,B 0,C 180,E1 7573.182,E2 7573.182} C_VEL
LIN {X 0,Y 397.765,Z 919.288,A -85,B 0,C 180,E1 7572.434,E2 7572.434} C_VEL
LIN {X 0,Y 405.133,Z 897.942,A -85,B 0,C 180,E1 7571.889,E2 7571.889} C_VEL
LIN {X 0,Y 411.336,Z 876.829,A -85,B 0,C 180,E1 7571.443,E2 7571.443} C_VEL
LIN {X 0,Y 417.058,Z 853.258,A -85,B 0,C 180,E1 7571.044,E2 7571.044} C_VEL
LIN {X 0,Y 422.34,Z 823.715,A -85,B 0,C 180,E1 7570.628,E2 7570.628} C_VEL
LIN {X 0,Y 430.124,Z 757.619,A -85,B 0,C 180,E1 7569.769,E2 7569.769} C_VEL
LIN {X 0,Y 440.71,Z 664.924,A -85,B 0,C 180,E1 7568.579,E2 7568.579} C_VEL
LIN {X 0,Y 439.928,Z 662.433,A -85,B 0,C 180,E1 7566.525,E2 7566.525} C_VEL
LIN {X 0,Y 439.463,Z 661.831,A -85,B 0,C 180,E1 7562.806,E2 7562.806} C_VEL
LIN {X 0,Y 440.03,Z 662.673,A -85,B 0,C 180,E1 7560.26,E2 7560.26} C_VEL
LIN {X 0,Y 440.702,Z 665.212,A -85,B 0,C 180,E1 7558.484,E2 7558.484} C_VEL
LIN {X 0,Y 438.927,Z 680.662,A -85,B 0,C 180,E1 7558.288,E2 7558.288} C_VEL
LIN {X 0,Y 437.954,Z 688.363,A -85,B 0,C 180,E1 7558.319,E2 7558.319} C_VEL
LIN {X 0,Y 435.041,Z 708.976,A -85,B 0,C 180,E1 7558.879,E2 7558.879} C_VEL
LIN {X 0,Y 434.215,Z 715.583,A -85,B 0,C 180,E1 7558.895,E2 7558.895} C_VEL
LIN {X 0,Y 421.587,Z 823.061,A -85,B 0,C 180,E1 7557.532,E2 7557.532} C_VEL
LIN {X 0,Y 416.859,Z 850.668,A -85,B 0,C 180,E1 7557.156,E2 7557.156} C_VEL
LIN {X 0,Y 410.413,Z 877.247,A -85,B 0,C 180,E1 7556.75,E2 7556.75} C_VEL
LIN {X 0,Y 404.016,Z 898.837,A -85,B 0,C 180,E1 7556.338,E2 7556.338} C_VEL
LIN {X 0,Y 396.493,Z 920.426,A -85,B 0,C 180,E1 7555.828,E2 7555.828} C_VEL
LIN {X 0,Y 385.921,Z 946.393,A -85,B 0,C 180,E1 7555.071,E2 7555.071} C_VEL
LIN {X 0,Y 374.846,Z 969.443,A -85,B 0,C 180,E1 7554.228,E2 7554.228} C_VEL
LIN {X 0,Y 364.381,Z 988.862,A -85,B 0,C 180,E1 7553.374,E2 7553.374} C_VEL
LIN {X 0,Y 353.763,Z 1006.693,A -85,B 0,C 180,E1 7552.439,E2 7552.439} C_VEL
LIN {X 0,Y 341.399,Z 1025.54,A -85,B 0,C 180,E1 7551.278,E2 7551.278} C_VEL
LIN {X 0,Y 325.298,Z 1047.719,A -85,B 0,C 180,E1 7549.6,E2 7549.6} C_VEL
LIN {X 0,Y 309.497,Z 1067.101,A -85,B 0,C 180,E1 7547.755,E2 7547.755} C_VEL
LIN {X 0,Y 295.8,Z 1082.577,A -85,B 0,C 180,E1 7545.955,E2 7545.955} C_VEL
LIN {X 0,Y 281.99,Z 1097.054,A -85,B 0,C 180,E1 7543.922,E2 7543.922} C_VEL
LIN {X 0,Y 266.085,Z 1112.56,A -85,B 0,C 180,E1 7541.249,E2 7541.249} C_VEL
LIN {X 0,Y 246.894,Z 1129.69,A -85,B 0,C 180,E1 7537.419,E2 7537.419} C_VEL
LIN {X 0,Y 231.827,Z 1142.198,A -85,B 0,C 180,E1 7533.778,E2 7533.778} C_VEL
LIN {X 0,Y 218.428,Z 1152.765,A -85,B 0,C 180,E1 7529.899,E2 7529.899} C_VEL
LIN {X 0,Y 203.015,Z 1164.492,A -85,B 0,C 180,E1 7524.353,E2 7524.353} C_VEL
LIN {X 0,Y 189.071,Z 1174.663,A -85,B 0,C 180,E1 7517.761,E2 7517.761} C_VEL
LIN {X 0,Y 179.307,Z 1181.873,A -85,B 0,C 180,E1 7511.573,E2 7511.573} C_VEL
LIN {X 0,Y 171.507,Z 1187.908,A -85,B 0,C 180,E1 7504.842,E2 7504.842} C_VEL
LIN {X 0,Y 165.795,Z 1192.812,A -85,B 0,C 180,E1 7497.669,E2 7497.669} C_VEL
LIN {X 0,Y 161.908,Z 1196.944,A -85,B 0,C 180,E1 7489.48,E2 7489.48} C_VEL
LIN {X 0,Y 160.146,Z 1199.998,A -85,B 0,C 180,E1 7480.431,E2 7480.431} C_VEL
LIN {X 0,Y 159.918,Z 1201.302,A -85,B 0,C 180,E1 7473.585,E2 7473.585} C_VEL
LIN {X 0,Y 159.914,Z 1201.684,A -85,B 0,C 180,E1 7467.491,E2 7467.491} C_VEL
LIN {X 0,Y 160.078,Z 1201.359,A -85,B 0,C 180,E1 7460.654,E2 7460.654} C_VEL
LIN {X 0,Y 161.638,Z 1199.774,A -85,B 0,C 180,E1 7451.611,E2 7451.611} C_VEL
LIN {X 0,Y 166.031,Z 1196.453,A -85,B 0,C 180,E1 7442.286,E2 7442.286} C_VEL
LIN {X 0,Y 172.151,Z 1192.575,A -85,B 0,C 180,E1 7434.901,E2 7434.901} C_VEL
LIN {X 0,Y 180.635,Z 1187.546,A -85,B 0,C 180,E1 7427.951,E2 7427.951} C_VEL
LIN {X 0,Y 191.322,Z 1181.335,A -85,B 0,C 180,E1 7421.585,E2 7421.585} C_VEL
LIN {X 0,Y 206.904,Z 1172.238,A -85,B 0,C 180,E1 7414.763,E2 7414.763} C_VEL
LIN {X 0,Y 224.238,Z 1161.417,A -85,B 0,C 180,E1 7409.08,E2 7409.08} C_VEL
LIN {X 0,Y 238.827,Z 1151.861,A -85,B 0,C 180,E1 7405.272,E2 7405.272} C_VEL
LIN {X 0,Y 254.321,Z 1141.086,A -85,B 0,C 180,E1 7401.902,E2 7401.902} C_VEL
LIN {X 0,Y 273.091,Z 1127.124,A -85,B 0,C 180,E1 7398.511,E2 7398.511} C_VEL
LIN {X 0,Y 292.685,Z 1111.041,A -85,B 0,C 180,E1 7395.559,E2 7395.559} C_VEL
LIN {X 0,Y 308.742,Z 1096.698,A -85,B 0,C 180,E1 7393.484,E2 7393.484} C_VEL
LIN {X 0,Y 323.949,Z 1082.001,A -85,B 0,C 180,E1 7391.754,E2 7391.754} C_VEL
LIN {X 0,Y 339.318,Z 1065.884,A -85,B 0,C 180,E1 7390.204,E2 7390.204} C_VEL
LIN {X 0,Y 356.983,Z 1045.586,A -85,B 0,C 180,E1 7388.622,E2 7388.622} C_VEL
LIN {X 0,Y 372.994,Z 1024.771,A -85,B 0,C 180,E1 7387.33,E2 7387.33} C_VEL
LIN {X 0,Y 385.64,Z 1006.652,A -85,B 0,C 180,E1 7386.401,E2 7386.401} C_VEL
LIN {X 0,Y 397.297,Z 988.232,A -85,B 0,C 180,E1 7385.613,E2 7385.613} C_VEL
LIN {X 0,Y 408.44,Z 968.683,A -85,B 0,C 180,E1 7384.911,E2 7384.911} C_VEL
LIN {X 0,Y 421.056,Z 943.596,A -85,B 0,C 180,E1 7384.174,E2 7384.174} C_VEL
LIN {X 0,Y 431.294,Z 919.487,A -85,B 0,C 180,E1 7383.611,E2 7383.611} C_VEL
LIN {X 0,Y 435.489,Z 908.683,A -85,B 0,C 180,E1 7383.394,E2 7383.394} C_VEL
LIN {X 0,Y 425.459,Z 933.511,A -85,B 0,C 180,E1 7382.834,E2 7382.834} C_VEL
LIN {X 0,Y 416.272,Z 953.314,A -85,B 0,C 180,E1 7382.291,E2 7382.291} C_VEL
LIN {X 0,Y 406.111,Z 972.757,A -85,B 0,C 180,E1 7381.657,E2 7381.657} C_VEL
LIN {X 0,Y 393.986,Z 993.459,A -85,B 0,C 180,E1 7380.853,E2 7380.853} C_VEL
LIN {X 0,Y 377.452,Z 1018.232,A -85,B 0,C 180,E1 7379.66,E2 7379.66} C_VEL
LIN {X 0,Y 363.836,Z 1036.383,A -85,B 0,C 180,E1 7378.583,E2 7378.583} C_VEL
LIN {X 0,Y 349.837,Z 1053.384,A -85,B 0,C 180,E1 7377.379,E2 7377.379} C_VEL
LIN {X 0,Y 334.79,Z 1070.099,A -85,B 0,C 180,E1 7375.943,E2 7375.943} C_VEL
LIN {X 0,Y 315.748,Z 1089.321,A -85,B 0,C 180,E1 7373.89,E2 7373.89} C_VEL
LIN {X 0,Y 298.079,Z 1105.339,A -85,B 0,C 180,E1 7371.701,E2 7371.701} C_VEL
LIN {X 0,Y 282.682,Z 1118.234,A -85,B 0,C 180,E1 7369.512,E2 7369.512} C_VEL
LIN {X 0,Y 266.877,Z 1130.518,A -85,B 0,C 180,E1 7366.929,E2 7366.929} C_VEL
LIN {X 0,Y 250.033,Z 1142.698,A -85,B 0,C 180,E1 7363.686,E2 7363.686} C_VEL
LIN {X 0,Y 229.447,Z 1156.384,A -85,B 0,C 180,E1 7358.795,E2 7358.795} C_VEL
LIN {X 0,Y 214.249,Z 1165.752,A -85,B 0,C 180,E1 7354.249,E2 7354.249} C_VEL
LIN {X 0,Y 201.116,Z 1173.487,A -85,B 0,C 180,E1 7349.325,E2 7349.325} C_VEL
LIN {X 0,Y 189.006,Z 1180.397,A -85,B 0,C 180,E1 7343.523,E2 7343.523} C_VEL
LIN {X 0,Y 176.76,Z 1187.376,A -85,B 0,C 180,E1 7335.457,E2 7335.457} C_VEL
LIN {X 0,Y 168.164,Z 1192.27,A -85,B 0,C 180,E1 7326.907,E2 7326.907} C_VEL
LIN {X 0,Y 163.465,Z 1195.249,A -85,B 0,C 180,E1 7319.297,E2 7319.297} C_VEL
LIN {X 0,Y 160.982,Z 1197.11,A -85,B 0,C 180,E1 7311.88,E2 7311.88} C_VEL
LIN {X 0,Y 160.103,Z 1197.993,A -85,B 0,C 180,E1 7305.206,E2 7305.206} C_VEL
LIN {X 0,Y 159.925,Z 1198.144,A -85,B 0,C 180,E1 7298.63,E2 7298.63} C_VEL
LIN {X 0,Y 159.937,Z 1197.65,A -85,B 0,C 180,E1 7292.508,E2 7292.508} C_VEL
LIN {X 0,Y 160.369,Z 1196.206,A -85,B 0,C 180,E1 7285.351,E2 7285.351} C_VEL
LIN {X 0,Y 162.381,Z 1193.255,A -85,B 0,C 180,E1 7276.831,E2 7276.831} C_VEL
LIN {X 0,Y 166.256,Z 1189.445,A -85,B 0,C 180,E1 7269.217,E2 7269.217} C_VEL
LIN {X 0,Y 171.92,Z 1184.776,A -85,B 0,C 180,E1 7262.273,E2 7262.273} C_VEL
LIN {X 0,Y 179.939,Z 1178.764,A -85,B 0,C 180,E1 7255.474,E2 7255.474} C_VEL
LIN {X 0,Y 191.439,Z 1170.533,A -85,B 0,C 180,E1 7248.448,E2 7248.448} C_VEL
LIN {X 0,Y 206.376,Z 1159.658,A -85,B 0,C 180,E1 7241.746,E2 7241.746} C_VEL
LIN {X 0,Y 219.546,Z 1149.792,A -85,B 0,C 180,E1 7237.157,E2 7237.157} C_VEL
LIN {X 0,Y 233.167,Z 1139.155,A -85,B 0,C 180,E1 7233.26,E2 7233.26} C_VEL
LIN {X 0,Y 248.424,Z 1126.585,A -85,B 0,C 180,E1 7229.616,E2 7229.616} C_VEL
LIN {X 0,Y 267.669,Z 1109.415,A -85,B 0,C 180,E1 7225.811,E2 7225.811} C_VEL
LIN {X 0,Y 282.122,Z 1095.405,A -85,B 0,C 180,E1 7223.378,E2 7223.378} C_VEL
LIN {X 0,Y 296.18,Z 1080.759,A -85,B 0,C 180,E1 7221.294,E2 7221.294} C_VEL
LIN {X 0,Y 310.582,Z 1064.541,A -85,B 0,C 180,E1 7219.395,E2 7219.395} C_VEL
LIN {X 0,Y 327.042,Z 1044.309,A -85,B 0,C 180,E1 7217.471,E2 7217.471} C_VEL
LIN {X 0,Y 342.035,Z 1023.544,A -85,B 0,C 180,E1 7215.898,E2 7215.898} C_VEL
LIN {X 0,Y 353.654,Z 1005.868,A -85,B 0,C 180,E1 7214.782,E2 7214.782} C_VEL
LIN {X 0,Y 364.893,Z 987.035,A -85,B 0,C 180,E1 7213.775,E2 7213.775} C_VEL
LIN {X 0,Y 375.877,Z 966.588,A -85,B 0,C 180,E1 7212.861,E2 7212.861} C_VEL
LIN {X 0,Y 388.471,Z 939.631,A -85,B 0,C 180,E1 7211.883,E2 7211.883} C_VEL
LIN {X 0,Y 397.074,Z 918.12,A -85,B 0,C 180,E1 7211.251,E2 7211.251} C_VEL
LIN {X 0,Y 404.281,Z 897.329,A -85,B 0,C 180,E1 7210.745,E2 7210.745} C_VEL
LIN {X 0,Y 410.605,Z 875.881,A -85,B 0,C 180,E1 7210.313,E2 7210.313} C_VEL
LIN {X 0,Y 417.073,Z 849.06,A -85,B 0,C 180,E1 7209.888,E2 7209.888} C_VEL
LIN {X 0,Y 421.696,Z 821.911,A -85,B 0,C 180,E1 7209.521,E2 7209.521} C_VEL
LIN {X 0,Y 437.077,Z 690.752,A -85,B 0,C 180,E1 7207.862,E2 7207.862} C_VEL
LIN {X 0,Y 439.289,Z 671.765,A -85,B 0,C 180,E1 7207.625,E2 7207.625} C_VEL
LIN {X 0,Y 438.909,Z 670.34,A -85,B 0,C 180,E1 7206.409,E2 7206.409} C_VEL
LIN {X 0,Y 438.482,Z 669.763,A -85,B 0,C 180,E1 7202.859,E2 7202.859} C_VEL
LIN {X 0,Y 439.003,Z 670.553,A -85,B 0,C 180,E1 7200.392,E2 7200.392} C_VEL
LIN {X 0,Y 439.269,Z 672.096,A -85,B 0,C 180,E1 7199.44,E2 7199.44} C_VEL
LIN {X 0,Y 434.215,Z 715.583,A -85,B 0,C 180,E1 7198.895,E2 7198.895} C_VEL
LIN {X 0,Y 433.243,Z 723.285,A -85,B 0,C 180,E1 7198.93,E2 7198.93} C_VEL
LIN {X 0,Y 430.374,Z 743.893,A -85,B 0,C 180,E1 7199.506,E2 7199.506} C_VEL
LIN {X 0,Y 429.55,Z 750.5,A -85,B 0,C 180,E1 7199.523,E2 7199.523} C_VEL
LIN {X 0,Y 420.683,Z 824.092,A -85,B 0,C 180,E1 7198.606,E2 7198.606} C_VEL
LIN {X 0,Y 415.534,Z 852.854,A -85,B 0,C 180,E1 7198.224,E2 7198.224} C_VEL
LIN {X 0,Y 409.414,Z 877.695,A -85,B 0,C 180,E1 7197.858,E2 7197.858} C_VEL
LIN {X 0,Y 403.083,Z 898.839,A -85,B 0,C 180,E1 7197.471,E2 7197.471} C_VEL
LIN {X 0,Y 395.49,Z 920.424,A -85,B 0,C 180,E1 7196.984,E2 7196.984} C_VEL
LIN {X 0,Y 385.078,Z 945.814,A -85,B 0,C 180,E1 7196.278,E2 7196.278} C_VEL
LIN {X 0,Y 373.728,Z 969.208,A -85,B 0,C 180,E1 7195.462,E2 7195.462} C_VEL
LIN {X 0,Y 362.907,Z 989.05,A -85,B 0,C 180,E1 7194.625,E2 7194.625} C_VEL
LIN {X 0,Y 352.062,Z 1007.006,A -85,B 0,C 180,E1 7193.719,E2 7193.719} C_VEL
LIN {X 0,Y 339.292,Z 1026.175,A -85,B 0,C 180,E1 7192.579,E2 7192.579} C_VEL
LIN {X 0,Y 322.039,Z 1049.368,A -85,B 0,C 180,E1 7190.864,E2 7190.864} C_VEL
LIN {X 0,Y 306.917,Z 1067.558,A -85,B 0,C 180,E1 7189.175,E2 7189.175} C_VEL
LIN {X 0,Y 292.465,Z 1083.538,A -85,B 0,C 180,E1 7187.361,E2 7187.361} C_VEL
LIN {X 0,Y 276.842,Z 1099.487,A -85,B 0,C 180,E1 7185.141,E2 7185.141} C_VEL
LIN {X 0,Y 257.181,Z 1117.763,A -85,B 0,C 180,E1 7181.879,E2 7181.879} C_VEL
LIN {X 0,Y 241.38,Z 1131.252,A -85,B 0,C 180,E1 7178.749,E2 7178.749} C_VEL
LIN {X 0,Y 226.707,Z 1143.013,A -85,B 0,C 180,E1 7175.303,E2 7175.303} C_VEL
LIN {X 0,Y 210.696,Z 1155.161,A -85,B 0,C 180,E1 7170.738,E2 7170.738} C_VEL
LIN {X 0,Y 193.868,Z 1167.189,A -85,B 0,C 180,E1 7164.574,E2 7164.574} C_VEL
LIN {X 0,Y 181.908,Z 1175.498,A -85,B 0,C 180,E1 7158.853,E2 7158.853} C_VEL
LIN {X 0,Y 171.787,Z 1182.578,A -85,B 0,C 180,E1 7152.466,E2 7152.466} C_VEL
LIN {X 0,Y 163.36,Z 1188.747,A -85,B 0,C 180,E1 7145.123,E2 7145.123} C_VEL
LIN {X 0,Y 156.297,Z 1194.652,A -85,B 0,C 180,E1 7135.379,E2 7135.379} C_VEL
LIN {X 0,Y 153.086,Z 1198.166,A -85,B 0,C 180,E1 7126.701,E2 7126.701} C_VEL
LIN {X 0,Y 152.057,Z 1200.229,A -85,B 0,C 180,E1 7119.08,E2 7119.08} C_VEL
LIN {X 0,Y 151.917,Z 1201.299,A -85,B 0,C 180,E1 7112.263,E2 7112.263} C_VEL
LIN {X 0,Y 151.916,Z 1201.644,A -85,B 0,C 180,E1 7105.848,E2 7105.848} C_VEL
LIN {X 0,Y 152.278,Z 1201.139,A -85,B 0,C 180,E1 7098.256,E2 7098.256} C_VEL
LIN {X 0,Y 154.596,Z 1199.125,A -85,B 0,C 180,E1 7088.649,E2 7088.649} C_VEL
LIN {X 0,Y 159.204,Z 1196.149,A -85,B 0,C 180,E1 7080.255,E2 7080.255} C_VEL
LIN {X 0,Y 166.145,Z 1192.163,A -85,B 0,C 180,E1 7072.568,E2 7072.568} C_VEL
LIN {X 0,Y 175.673,Z 1186.945,A -85,B 0,C 180,E1 7065.355,E2 7065.355} C_VEL
LIN {X 0,Y 189.816,Z 1179.308,A -85,B 0,C 180,E1 7057.803,E2 7057.803} C_VEL
LIN {X 0,Y 206.902,Z 1169.528,A -85,B 0,C 180,E1 7051.201,E2 7051.201} C_VEL
LIN {X 0,Y 221.757,Z 1160.633,A -85,B 0,C 180,E1 7046.781,E2 7046.781} C_VEL
LIN {X 0,Y 236.942,Z 1150.996,A -85,B 0,C 180,E1 7043.085,E2 7043.085} C_VEL
LIN {X 0,Y 253.794,Z 1139.572,A -85,B 0,C 180,E1 7039.683,E2 7039.683} C_VEL
LIN {X 0,Y 275.717,Z 1123.331,A -85,B 0,C 180,E1 7036.056,E2 7036.056} C_VEL
LIN {X 0,Y 293.234,Z 1109.041,A -85,B 0,C 180,E1 7033.645,E2 7033.645} C_VEL
LIN {X 0,Y 308.928,Z 1095.172,A -85,B 0,C 180,E1 7031.766,E2 7031.766} C_VEL
LIN {X 0,Y 324.96,Z 1079.806,A -85,B 0,C 180,E1 7030.07,E2 7030.07} C_VEL
LIN {X 0,Y 344.272,Z 1059.456,A -85,B 0,C 180,E1 7028.284,E2 7028.284} C_VEL
LIN {X 0,Y 360.595,Z 1040.112,A -85,B 0,C 180,E1 7026.946,E2 7026.946} C_VEL
LIN {X 0,Y 373.968,Z 1022.701,A -85,B 0,C 180,E1 7025.961,E2 7025.961} C_VEL
LIN {X 0,Y 386.476,Z 1004.801,A -85,B 0,C 180,E1 7025.102,E2 7025.102} C_VEL
LIN {X 0,Y 399.077,Z 984.846,A -85,B 0,C 180,E1 7024.311,E2 7024.311} C_VEL
LIN {X 0,Y 413.696,Z 958.399,A -85,B 0,C 180,E1 7023.463,E2 7023.463} C_VEL
LIN {X 0,Y 415.307,Z 955.152,A -85,B 0,C 180,E1 7023.359,E2 7023.359} C_VEL
LIN {X 0,Y 404.118,Z 976.118,A -85,B 0,C 180,E1 7022.695,E2 7022.695} C_VEL
LIN {X 0,Y 388.617,Z 1001.435,A -85,B 0,C 180,E1 7021.71,E2 7021.71} C_VEL
LIN {X 0,Y 374.97,Z 1021.068,A -85,B 0,C 180,E1 7020.764,E2 7020.764} C_VEL
LIN {X 0,Y 361.95,Z 1038.06,A -85,B 0,C 180,E1 7019.781,E2 7019.781} C_VEL
LIN {X 0,Y 347.553,Z 1055.198,A -85,B 0,C 180,E1 7018.603,E2 7018.603} C_VEL
LIN {X 0,Y 329.423,Z 1074.816,A -85,B 0,C 180,E1 7016.938,E2 7016.938} C_VEL
LIN {X 0,Y 311.022,Z 1092.511,A -85,B 0,C 180,E1 7015.02,E2 7015.02} C_VEL
LIN {X 0,Y 295.084,Z 1106.591,A -85,B 0,C 180,E1 7013.118,E2 7013.118} C_VEL
LIN {X 0,Y 278.974,Z 1119.722,A -85,B 0,C 180,E1 7010.926,E2 7010.926} C_VEL
LIN {X 0,Y 260.645,Z 1133.513,A -85,B 0,C 180,E1 7008.015,E2 7008.015} C_VEL
LIN {X 0,Y 240.042,Z 1147.58,A -85,B 0,C 180,E1 7004.043,E2 7004.043} C_VEL
LIN {X 0,Y 223.346,Z 1158.066,A -85,B 0,C 180,E1 7000.07,E2 7000.07} C_VEL
LIN {X 0,Y 208.429,Z 1166.856,A -85,B 0,C 180,E1 6995.707,E2 6995.707} C_VEL
LIN {X 0,Y 193.571,Z 1175.177,A -85,B 0,C 180,E1 6990.201,E2 6990.201} C_VEL
LIN {X 0,Y 177.454,Z 1183.756,A -85,B 0,C 180,E1 6982.076,E2 6982.076} C_VEL
LIN {X 0,Y 167.394,Z 1189.019,A -85,B 0,C 180,E1 6974.815,E2 6974.815} C_VEL
LIN {X 0,Y 160.168,Z 1192.913,A -85,B 0,C 180,E1 6967.267,E2 6967.267} C_VEL
LIN {X 0,Y 155.363,Z 1195.73,A -85,B 0,C 180,E1 6959.282,E2 6959.282} C_VEL
LIN {X 0,Y 152.879,Z 1197.431,A -85,B 0,C 180,E1 6951.485,E2 6951.485} C_VEL
LIN {X 0,Y 152.054,Z 1198.156,A -85,B 0,C 180,E1 6944.47,E2 6944.47} C_VEL
LIN {X 0,Y 151.922,Z 1198.197,A -85,B 0,C 180,E1 6938.325,E2 6938.325} C_VEL
LIN {X 0,Y 151.948,Z 1197.638,A -85,B 0,C 180,E1 6931.886,E2 6931.886} C_VEL
LIN {X 0,Y 152.487,Z 1196.132,A -85,B 0,C 180,E1 6924.356,E2 6924.356} C_VEL
LIN {X 0,Y 154.712,Z 1193.272,A -85,B 0,C 180,E1 6915.784,E2 6915.784} C_VEL
LIN {X 0,Y 158.99,Z 1189.443,A -85,B 0,C 180,E1 6907.832,E2 6907.832} C_VEL
LIN {X 0,Y 165.141,Z 1184.753,A -85,B 0,C 180,E1 6900.632,E2 6900.632} C_VEL
LIN {X 0,Y 173.651,Z 1178.788,A -85,B 0,C 180,E1 6893.72,E2 6893.72} C_VEL
LIN {X 0,Y 185.975,Z 1170.466,A -85,B 0,C 180,E1 6886.515,E2 6886.515} C_VEL
LIN {X 0,Y 201.052,Z 1159.991,A -85,B 0,C 180,E1 6880.016,E2 6880.016} C_VEL
LIN {X 0,Y 214.735,Z 1150.154,A -85,B 0,C 180,E1 6875.429,E2 6875.429} C_VEL
LIN {X 0,Y 228.814,Z 1139.547,A -85,B 0,C 180,E1 6871.56,E2 6871.56} C_VEL
LIN {X 0,Y 244.518,Z 1127.005,A -85,B 0,C 180,E1 6867.964,E2 6867.964} C_VEL
LIN {X 0,Y 264.246,Z 1109.905,A -85,B 0,C 180,E1 6864.232,E2 6864.232} C_VEL
LIN {X 0,Y 279.851,Z 1095.105,A -85,B 0,C 180,E1 6861.732,E2 6861.732} C_VEL
LIN {X 0,Y 294.203,Z 1080.413,A -85,B 0,C 180,E1 6859.714,E2 6859.714} C_VEL
LIN {X 0,Y 308.876,Z 1064.151,A -85,B 0,C 180,E1 6857.88,E2 6857.88} C_VEL
LIN {X 0,Y 326.497,Z 1042.631,A -85,B 0,C 180,E1 6855.933,E2 6855.933} C_VEL
LIN {X 0,Y 340.831,Z 1022.999,A -85,B 0,C 180,E1 6854.515,E2 6854.515} C_VEL
LIN {X 0,Y 352.637,Z 1005.222,A -85,B 0,C 180,E1 6853.445,E2 6853.445} C_VEL
LIN {X 0,Y 364.045,Z 986.268,A -85,B 0,C 180,E1 6852.477,E2 6852.477} C_VEL
LIN {X 0,Y 376.857,Z 962.5,A -85,B 0,C 180,E1 6851.478,E2 6851.478} C_VEL
LIN {X 0,Y 388.129,Z 937.972,A -85,B 0,C 180,E1 6850.65,E2 6850.65} C_VEL
LIN {X 0,Y 396.546,Z 916.972,A -85,B 0,C 180,E1 6850.065,E2 6850.065} C_VEL
LIN {X 0,Y 403.825,Z 895.98,A -85,B 0,C 180,E1 6849.581,E2 6849.581} C_VEL
LIN {X 0,Y 410.745,Z 872.352,A -85,B 0,C 180,E1 6849.136,E2 6849.136} C_VEL
LIN {X 0,Y 417.321,Z 843.437,A -85,B 0,C 180,E1 6848.716,E2 6848.716} C_VEL
LIN {X 0,Y 421.175,Z 820.266,A -85,B 0,C 180,E1 6848.414,E2 6848.414} C_VEL
LIN {X 0,Y 437.998,Z 678.512,A -85,B 0,C 180,E1 6846.656,E2 6846.656} C_VEL
LIN {X 0,Y 437.481,Z 677.673,A -85,B 0,C 180,E1 6843.407,E2 6843.407} C_VEL
LIN {X 0,Y 438.005,Z 678.594,A -85,B 0,C 180,E1 6840.407,E2 6840.407} C_VEL
LIN {X 0,Y 429.55,Z 750.5,A -85,B 0,C 180,E1 6839.523,E2 6839.523} C_VEL
LIN {X 0,Y 428.582,Z 758.199,A -85,B 0,C 180,E1 6839.559,E2 6839.559} C_VEL
LIN {X 0,Y 425.761,Z 778.8,A -85,B 0,C 180,E1 6840.148,E2 6840.148} C_VEL
LIN {X 0,Y 424.937,Z 785.408,A -85,B 0,C 180,E1 6840.169,E2 6840.169} C_VEL
LIN {X 0,Y 419.245,Z 829.986,A -85,B 0,C 180,E1 6839.623,E2 6839.623} C_VEL
LIN {X 0,Y 413.817,Z 857.339,A -85,B 0,C 180,E1 6839.267,E2 6839.267} C_VEL
LIN {X 0,Y 408.227,Z 879.343,A -85,B 0,C 180,E1 6838.953,E2 6838.953} C_VEL
LIN {X 0,Y 401.687,Z 900.714,A -85,B 0,C 180,E1 6838.574,E2 6838.574} C_VEL
LIN {X 0,Y 392.489,Z 926.148,A -85,B 0,C 180,E1 6838.008,E2 6838.008} C_VEL
LIN {X 0,Y 381.369,Z 951.578,A -85,B 0,C 180,E1 6837.295,E2 6837.295} C_VEL
LIN {X 0,Y 371.39,Z 971.609,A -85,B 0,C 180,E1 6836.604,E2 6836.604} C_VEL
LIN {X 0,Y 360.902,Z 990.448,A -85,B 0,C 180,E1 6835.832,E2 6835.832} C_VEL
LIN {X 0,Y 348.894,Z 1009.898,A -85,B 0,C 180,E1 6834.874,E2 6834.874} C_VEL
LIN {X 0,Y 332.141,Z 1034.015,A -85,B 0,C 180,E1 6833.418,E2 6833.418} C_VEL
LIN {X 0,Y 317.872,Z 1052.314,A -85,B 0,C 180,E1 6832.044,E2 6832.044} C_VEL
LIN {X 0,Y 304.068,Z 1068.535,A -85,B 0,C 180,E1 6830.567,E2 6830.567} C_VEL
LIN {X 0,Y 289.455,Z 1084.346,A -85,B 0,C 180,E1 6828.817,E2 6828.817} C_VEL
LIN {X 0,Y 271.575,Z 1102.156,A -85,B 0,C 180,E1 6826.371,E2 6826.371} C_VEL
LIN {X 0,Y 253.438,Z 1118.387,A -85,B 0,C 180,E1 6823.47,E2 6823.47} C_VEL
LIN {X 0,Y 238.447,Z 1130.858,A -85,B 0,C 180,E1 6820.642,E2 6820.642} C_VEL
LIN {X 0,Y 223.305,Z 1142.649,A -85,B 0,C 180,E1 6817.275,E2 6817.275} C_VEL
LIN {X 0,Y 207.758,Z 1154.049,A -85,B 0,C 180,E1 6813.102,E2 6813.102} C_VEL
LIN {X 0,Y 189.091,Z 1166.907,A -85,B 0,C 180,E1 6806.663,E2 6806.663} C_VEL
LIN {X 0,Y 176.48,Z 1175.241,A -85,B 0,C 180,E1 6800.912,E2 6800.912} C_VEL
LIN {X 0,Y 166.156,Z 1182.036,A -85,B 0,C 180,E1 6794.753,E2 6794.753} C_VEL
LIN {X 0,Y 157.338,Z 1188.018,A -85,B 0,C 180,E1 6787.594,E2 6787.594} C_VEL
LIN {X 0,Y 150.268,Z 1193.294,A -85,B 0,C 180,E1 6779.06,E2 6779.06} C_VEL
LIN {X 0,Y 145.494,Z 1197.793,A -85,B 0,C 180,E1 6768.428,E2 6768.428} C_VEL
LIN {X 0,Y 144.083,Z 1200.111,A -85,B 0,C 180,E1 6759.587,E2 6759.587} C_VEL
LIN {X 0,Y 143.917,Z 1201.202,A -85,B 0,C 180,E1 6752.389,E2 6752.389} C_VEL
LIN {X 0,Y 143.915,Z 1201.553,A -85,B 0,C 180,E1 6746.016,E2 6746.016} C_VEL
LIN {X 0,Y 144.255,Z 1201.128,A -85,B 0,C 180,E1 6738.404,E2 6738.404} C_VEL
LIN {X 0,Y 146.611,Z 1199.35,A -85,B 0,C 180,E1 6728.391,E2 6728.391} C_VEL
LIN {X 0,Y 152.016,Z 1196.157,A -85,B 0,C 180,E1 6718.769,E2 6718.769} C_VEL
LIN {X 0,Y 159.602,Z 1192.167,A -85,B 0,C 180,E1 6710.748,E2 6710.748} C_VEL
LIN {X 0,Y 169.582,Z 1187.089,A -85,B 0,C 180,E1 6703.514,E2 6703.514} C_VEL
LIN {X 0,Y 182.959,Z 1180.263,A -85,B 0,C 180,E1 6696.549,E2 6696.549} C_VEL
LIN {X 0,Y 201.984,Z 1170.027,A -85,B 0,C 180,E1 6689.398,E2 6689.398} C_VEL
LIN {X 0,Y 218.108,Z 1160.76,A -85,B 0,C 180,E1 6684.814,E2 6684.814} C_VEL
LIN {X 0,Y 233.79,Z 1151.152,A -85,B 0,C 180,E1 6681.2,E2 6681.2} C_VEL
LIN {X 0,Y 251.109,Z 1139.755,A -85,B 0,C 180,E1 6677.891,E2 6677.891} C_VEL
LIN {X 0,Y 272.658,Z 1124.265,A -85,B 0,C 180,E1 6674.51,E2 6674.51} C_VEL
LIN {X 0,Y 291.395,Z 1109.317,A -85,B 0,C 180,E1 6672.065,E2 6672.065} C_VEL
LIN {X 0,Y 306.913,Z 1095.89,A -85,B 0,C 180,E1 6670.312,E2 6670.312} C_VEL
LIN {X 0,Y 322.692,Z 1081.078,A -85,B 0,C 180,E1 6668.73,E2 6668.73} C_VEL
LIN {X 0,Y 339.65,Z 1063.699,A -85,B 0,C 180,E1 6667.228,E2 6667.228} C_VEL
LIN {X 0,Y 358.744,Z 1041.804,A -85,B 0,C 180,E1 6665.736,E2 6665.736} C_VEL
LIN {X 0,Y 373.216,Z 1023.253,A -85,B 0,C 180,E1 6664.728,E2 6664.728} C_VEL
LIN {X 0,Y 385.844,Z 1005.416,A -85,B 0,C 180,E1 6663.913,E2 6663.913} C_VEL
LIN {X 0,Y 395.256,Z 990.898,A -85,B 0,C 180,E1 6663.336,E2 6663.336} C_VEL
LIN {X 0,Y 380.614,Z 1013.078,A -85,B 0,C 180,E1 6662.409,E2 6662.409} C_VEL
LIN {X 0,Y 364.037,Z 1035.024,A -85,B 0,C 180,E1 6661.275,E2 6661.275} C_VEL
LIN {X 0,Y 349.384,Z 1052.511,A -85,B 0,C 180,E1 6660.164,E2 6660.164} C_VEL
LIN {X 0,Y 335.007,Z 1068.182,A -85,B 0,C 180,E1 6658.958,E2 6658.958} C_VEL
LIN {X 0,Y 319.106,Z 1084.052,A -85,B 0,C 180,E1 6657.486,E2 6657.486} C_VEL
LIN {X 0,Y 297.986,Z 1103.109,A -85,B 0,C 180,E1 6655.237,E2 6655.237} C_VEL
LIN {X 0,Y 280.041,Z 1117.656,A -85,B 0,C 180,E1 6653.011,E2 6653.011} C_VEL
LIN {X 0,Y 263.328,Z 1130.119,A -85,B 0,C 180,E1 6650.603,E2 6650.603} C_VEL
LIN {X 0,Y 246.564,Z 1141.67,A -85,B 0,C 180,E1 6647.767,E2 6647.767} C_VEL
LIN {X 0,Y 226.185,Z 1154.643,A -85,B 0,C 180,E1 6643.565,E2 6643.565} C_VEL
LIN {X 0,Y 207.243,Z 1165.486,A -85,B 0,C 180,E1 6638.613,E2 6638.613} C_VEL
LIN {X 0,Y 192.764,Z 1173.277,A -85,B 0,C 180,E1 6633.81,E2 6633.81} C_VEL
LIN {X 0,Y 179.149,Z 1180.241,A -85,B 0,C 180,E1 6628.031,E2 6628.031} C_VEL
LIN {X 0,Y 165.502,Z 1187.053,A -85,B 0,C 180,E1 6620.108,E2 6620.108} C_VEL
LIN {X 0,Y 154.727,Z 1192.276,A -85,B 0,C 180,E1 6610.743,E2 6610.743} C_VEL
LIN {X 0,Y 148.553,Z 1195.451,A -85,B 0,C 180,E1 6601.995,E2 6601.995} C_VEL
LIN {X 0,Y 145.414,Z 1197.284,A -85,B 0,C 180,E1 6593.934,E2 6593.934} C_VEL
LIN {X 0,Y 144.201,Z 1198.17,A -85,B 0,C 180,E1 6586.516,E2 6586.516} C_VEL
LIN {X 0,Y 143.93,Z 1198.335,A -85,B 0,C 180,E1 6579.429,E2 6579.429} C_VEL
LIN {X 0,Y 143.933,Z 1197.898,A -85,B 0,C 180,E1 6572.787,E2 6572.787} C_VEL
LIN {X 0,Y 144.418,Z 1196.504,A -85,B 0,C 180,E1 6564.836,E2 6564.836} C_VEL
LIN {X 0,Y 146.859,Z 1193.52,A -85,B 0,C 180,E1 6555.198,E2 6555.198} C_VEL
LIN {X 0,Y 151.545,Z 1189.641,A -85,B 0,C 180,E1 6546.68,E2 6546.68} C_VEL
LIN {X 0,Y 158.136,Z 1184.978,A -85,B 0,C 180,E1 6539.193,E2 6539.193} C_VEL
LIN {X 0,Y 166.889,Z 1179.223,A -85,B 0,C 180,E1 6532.266,E2 6532.266} C_VEL
LIN {X 0,Y 178.484,Z 1171.778,A -85,B 0,C 180,E1 6525.554,E2 6525.554} C_VEL
LIN {X 0,Y 195.276,Z 1160.772,A -85,B 0,C 180,E1 6518.428,E2 6518.428} C_VEL
LIN {X 0,Y 210.128,Z 1150.515,A -85,B 0,C 180,E1 6513.622,E2 6513.622} C_VEL
LIN {X 0,Y 224.67,Z 1139.936,A -85,B 0,C 180,E1 6509.795,E2 6509.795} C_VEL
LIN {X 0,Y 240.031,Z 1128.047,A -85,B 0,C 180,E1 6506.416,E2 6506.416} C_VEL
LIN {X 0,Y 258.977,Z 1112.27,A -85,B 0,C 180,E1 6502.952,E2 6502.952} C_VEL
LIN {X 0,Y 276.963,Z 1095.624,A -85,B 0,C 180,E1 6500.18,E2 6500.18} C_VEL
LIN {X 0,Y 291.584,Z 1080.972,A -85,B 0,C 180,E1 6498.223,E2 6498.223} C_VEL
LIN {X 0,Y 306.502,Z 1064.753,A -85,B 0,C 180,E1 6496.449,E2 6496.449} C_VEL
LIN {X 0,Y 323.939,Z 1043.929,A -85,B 0,C 180,E1 6494.617,E2 6494.617} C_VEL
LIN {X 0,Y 339.371,Z 1023.106,A -85,B 0,C 180,E1 6493.165,E2 6493.165} C_VEL
LIN {X 0,Y 351.263,Z 1005.433,A -85,B 0,C 180,E1 6492.146,E2 6492.146} C_VEL
LIN {X 0,Y 362.41,Z 987.17,A -85,B 0,C 180,E1 6491.248,E2 6491.248} C_VEL
LIN {X 0,Y 374.069,Z 965.918,A -85,B 0,C 180,E1 6490.381,E2 6490.381} C_VEL
LIN {X 0,Y 386.745,Z 939.17,A -85,B 0,C 180,E1 6489.498,E2 6489.498} C_VEL
LIN {X 0,Y 395.242,Z 918.306,A -85,B 0,C 180,E1 6488.938,E2 6488.938} C_VEL
LIN {X 0,Y 402.587,Z 897.499,A -85,B 0,C 180,E1 6488.474,E2 6488.474} C_VEL
LIN {X 0,Y 409.061,Z 875.925,A -85,B 0,C 180,E1 6488.077,E2 6488.077} C_VEL
LIN {X 0,Y 415.674,Z 848.872,A -85,B 0,C 180,E1 6487.686,E2 6487.686} C_VEL
LIN {X 0,Y 420.351,Z 821.895,A -85,B 0,C 180,E1 6487.344,E2 6487.344} C_VEL
LIN {X 0,Y 436.746,Z 685.983,A -85,B 0,C 180,E1 6485.686,E2 6485.686} C_VEL
LIN {X 0,Y 436.573,Z 685.748,A -85,B 0,C 180,E1 6482.363,E2 6482.363} C_VEL
LIN {X 0,Y 436.737,Z 686.175,A -85,B 0,C 180,E1 6481.366,E2 6481.366} C_VEL
LIN {X 0,Y 424.937,Z 785.408,A -85,B 0,C 180,E1 6480.169,E2 6480.169} C_VEL
LIN {X 0,Y 423.977,Z 793.105,A -85,B 0,C 180,E1 6480.21,E2 6480.21} C_VEL
LIN {X 0,Y 421.143,Z 813.686,A -85,B 0,C 180,E1 6480.814,E2 6480.814} C_VEL
LIN {X 0,Y 420.157,Z 820.277,A -85,B 0,C 180,E1 6480.836,E2 6480.836} C_VEL
LIN {X 0,Y 416.352,Z 842.926,A -85,B 0,C 180,E1 6480.557,E2 6480.557} C_VEL
LIN {X 0,Y 410.13,Z 870.582,A -85,B 0,C 180,E1 6480.204,E2 6480.204} C_VEL
LIN {X 0,Y 402.693,Z 895.761,A -85,B 0,C 180,E1 6479.807,E2 6479.807} C_VEL
LIN {X 0,Y 395.24,Z 916.999,A -85,B 0,C 180,E1 6479.388,E2 6479.388} C_VEL
LIN {X 0,Y 387.014,Z 937.294,A -85,B 0,C 180,E1 6478.903,E2 6478.903} C_VEL
LIN {X 0,Y 376.748,Z 959.493,A -85,B 0,C 180,E1 6478.258,E2 6478.258} C_VEL
LIN {X 0,Y 362.735,Z 985.592,A -85,B 0,C 180,E1 6477.314,E2 6477.314} C_VEL
LIN {X 0,Y 351.118,Z 1004.654,A -85,B 0,C 180,E1 6476.462,E2 6476.462} C_VEL
LIN {X 0,Y 338.991,Z 1022.653,A -85,B 0,C 180,E1 6475.509,E2 6475.509} C_VEL
LIN {X 0,Y 325.722,Z 1040.576,A -85,B 0,C 180,E1 6474.363,E2 6474.363} C_VEL
LIN {X 0,Y 308.826,Z 1061.301,A -85,B 0,C 180,E1 6472.746,E2 6472.746} C_VEL
LIN {X 0,Y 291.635,Z 1080.006,A -85,B 0,C 180,E1 6470.892,E2 6470.892} C_VEL
LIN {X 0,Y 276.96,Z 1094.684,A -85,B 0,C 180,E1 6469.097,E2 6469.097} C_VEL
LIN {X 0,Y 261.686,Z 1108.807,A -85,B 0,C 180,E1 6466.971,E2 6466.971} C_VEL
LIN {X 0,Y 245.869,Z 1122.353,A -85,B 0,C 180,E1 6464.431,E2 6464.431} C_VEL
LIN {X 0,Y 226.146,Z 1137.937,A -85,B 0,C 180,E1 6460.634,E2 6460.634} C_VEL
LIN {X 0,Y 208.389,Z 1150.701,A -85,B 0,C 180,E1 6456.409,E2 6456.409} C_VEL
LIN {X 0,Y 193.58,Z 1160.741,A -85,B 0,C 180,E1 6452.034,E2 6452.034} C_VEL
LIN {X 0,Y 179.324,Z 1169.956,A -85,B 0,C 180,E1 6446.757,E2 6446.757} C_VEL
LIN {X 0,Y 163.952,Z 1179.622,A -85,B 0,C 180,E1 6439.131,E2 6439.131} C_VEL
LIN {X 0,Y 152.434,Z 1186.764,A -85,B 0,C 180,E1 6430.99,E2 6430.99} C_VEL
LIN {X 0,Y 144.805,Z 1191.836,A -85,B 0,C 180,E1 6423.058,E2 6423.058} C_VEL
LIN {X 0,Y 139.805,Z 1195.642,A -85,B 0,C 180,E1 6414.958,E2 6414.958} C_VEL
LIN {X 0,Y 137.08,Z 1198.354,A -85,B 0,C 180,E1 6406.963,E2 6406.963} C_VEL
LIN {X 0,Y 136.065,Z 1200.132,A -85,B 0,C 180,E1 6399.303,E2 6399.303} C_VEL
LIN {X 0,Y 135.918,Z 1201.127,A -85,B 0,C 180,E1 6392.108,E2 6392.108} C_VEL
LIN {X 0,Y 135.92,Z 1201.475,A -85,B 0,C 180,E1 6385.359,E2 6385.359} C_VEL
LIN {X 0,Y 136.423,Z 1200.999,A -85,B 0,C 180,E1 6376.868,E2 6376.868} C_VEL
LIN {X 0,Y 139.35,Z 1199.08,A -85,B 0,C 180,E1 6366.309,E2 6366.309} C_VEL
LIN {X 0,Y 145.038,Z 1196.112,A -85,B 0,C 180,E1 6357.002,E2 6357.002} C_VEL
LIN {X 0,Y 153.232,Z 1192.17,A -85,B 0,C 180,E1 6348.774,E2 6348.774} C_VEL
LIN {X 0,Y 163.933,Z 1187.116,A -85,B 0,C 180,E1 6341.392,E2 6341.392} C_VEL
LIN {X 0,Y 177.452,Z 1180.615,A -85,B 0,C 180,E1 6334.65,E2 6334.65} C_VEL
LIN {X 0,Y 197.276,Z 1170.529,A -85,B 0,C 180,E1 6327.507,E2 6327.507} C_VEL
LIN {X 0,Y 214.724,Z 1160.889,A -85,B 0,C 180,E1 6322.783,E2 6322.783} C_VEL
LIN {X 0,Y 231.337,Z 1151.037,A -85,B 0,C 180,E1 6319.177,E2 6319.177} C_VEL
LIN {X 0,Y 248.673,Z 1139.939,A -85,B 0,C 180,E1 6316.062,E2 6316.062} C_VEL
LIN {X 0,Y 269.803,Z 1125.199,A -85,B 0,C 180,E1 6312.93,E2 6312.93} C_VEL
LIN {X 0,Y 289.78,Z 1109.601,A -85,B 0,C 180,E1 6310.467,E2 6310.467} C_VEL
LIN {X 0,Y 305.549,Z 1096.212,A -85,B 0,C 180,E1 6308.795,E2 6308.795} C_VEL
LIN {X 0,Y 321.551,Z 1081.438,A -85,B 0,C 180,E1 6307.288,E2 6307.288} C_VEL
LIN {X 0,Y 337.761,Z 1065.098,A -85,B 0,C 180,E1 6305.934,E2 6305.934} C_VEL
LIN {X 0,Y 357.055,Z 1043.497,A -85,B 0,C 180,E1 6304.513,E2 6304.513} C_VEL
LIN {X 0,Y 372.638,Z 1023.806,A -85,B 0,C 180,E1 6303.492,E2 6303.492} C_VEL
LIN {X 0,Y 375.193,Z 1020.379,A -85,B 0,C 180,E1 6303.316,E2 6303.316} C_VEL
LIN {X 0,Y 362.284,Z 1036.979,A -85,B 0,C 180,E1 6302.47,E2 6302.47} C_VEL
LIN {X 0,Y 348.061,Z 1053.656,A -85,B 0,C 180,E1 6301.451,E2 6301.451} C_VEL
LIN {X 0,Y 332.955,Z 1069.821,A -85,B 0,C 180,E1 6300.254,E2 6300.254} C_VEL
LIN {X 0,Y 313.686,Z 1088.572,A -85,B 0,C 180,E1 6298.539,E2 6298.539} C_VEL
LIN {X 0,Y 294.482,Z 1105.16,A -85,B 0,C 180,E1 6296.579,E2 6296.579} C_VEL
LIN {X 0,Y 277.218,Z 1118.801,A -85,B 0,C 180,E1 6294.54,E2 6294.54} C_VEL
LIN {X 0,Y 260.352,Z 1131.055,A -85,B 0,C 180,E1 6292.232,E2 6292.232} C_VEL
LIN {X 0,Y 241.29,Z 1143.794,A -85,B 0,C 180,E1 6289.136,E2 6289.136} C_VEL
LIN {X 0,Y 219.667,Z 1156.812,A -85,B 0,C 180,E1 6284.787,E2 6284.787} C_VEL
LIN {X 0,Y 202.638,Z 1166.181,A -85,B 0,C 180,E1 6280.464,E2 6280.464} C_VEL
LIN {X 0,Y 187.619,Z 1173.892,A -85,B 0,C 180,E1 6275.684,E2 6275.684} C_VEL
LIN {X 0,Y 172.14,Z 1181.397,A -85,B 0,C 180,E1 6269.276,E2 6269.276} C_VEL
LIN {X 0,Y 156.511,Z 1188.557,A -85,B 0,C 180,E1 6260.05,E2 6260.05} C_VEL
LIN {X 0,Y 147.045,Z 1192.823,A -85,B 0,C 180,E1 6251.583,E2 6251.583} C_VEL
LIN {X 0,Y 140.978,Z 1195.675,A -85,B 0,C 180,E1 6243.1,E2 6243.1} C_VEL
LIN {X 0,Y 137.577,Z 1197.438,A -85,B 0,C 180,E1 6234.703,E2 6234.703} C_VEL
LIN {X 0,Y 136.207,Z 1198.29,A -85,B 0,C 180,E1 6226.636,E2 6226.636} C_VEL
LIN {X 0,Y 135.929,Z 1198.399,A -85,B 0,C 180,E1 6219.313,E2 6219.313} C_VEL
LIN {X 0,Y 135.936,Z 1197.954,A -85,B 0,C 180,E1 6212.529,E2 6212.529} C_VEL
LIN {X 0,Y 136.447,Z 1196.652,A -85,B 0,C 180,E1 6204.534,E2 6204.534} C_VEL
LIN {X 0,Y 139.18,Z 1193.619,A -85,B 0,C 180,E1 6194.158,E2 6194.158} C_VEL
LIN {X 0,Y 144.352,Z 1189.704,A -85,B 0,C 180,E1 6185.15,E2 6185.15} C_VEL
LIN {X 0,Y 151.629,Z 1184.953,A -85,B 0,C 180,E1 6177.268,E2 6177.268} C_VEL
LIN {X 0,Y 160.958,Z 1179.221,A -85,B 0,C 180,E1 6170.221,E2 6170.221} C_VEL
LIN {X 0,Y 173.362,Z 1171.709,A -85,B 0,C 180,E1 6163.39,E2 6163.39} C_VEL
LIN {X 0,Y 191.676,Z 1160.205,A -85,B 0,C 180,E1 6156.047,E2 6156.047} C_VEL
LIN {X 0,Y 206.487,Z 1150.358,A -85,B 0,C 180,E1 6151.532,E2 6151.532} C_VEL
LIN {X 0,Y 221.521,Z 1139.764,A -85,B 0,C 180,E1 6147.79,E2 6147.79} C_VEL
LIN {X 0,Y 237.344,Z 1127.843,A -85,B 0,C 180,E1 6144.503,E2 6144.503} C_VEL
LIN {X 0,Y 257.182,Z 1111.628,A -85,B 0,C 180,E1 6141.084,E2 6141.084} C_VEL
LIN {X 0,Y 274.282,Z 1096.143,A -85,B 0,C 180,E1 6138.596,E2 6138.596} C_VEL
LIN {X 0,Y 289.165,Z 1081.531,A -85,B 0,C 180,E1 6136.707,E2 6136.707} C_VEL
LIN {X 0,Y 303.469,Z 1066.297,A -85,B 0,C 180,E1 6135.088,E2 6135.088} C_VEL
LIN {X 0,Y 318.358,Z 1049.019,A -85,B 0,C 180,E1 6133.583,E2 6133.583} C_VEL
LIN {X 0,Y 336.256,Z 1025.828,A -85,B 0,C 180,E1 6131.964,E2 6131.964} C_VEL
LIN {X 0,Y 349.468,Z 1006.576,A -85,B 0,C 180,E1 6130.885,E2 6130.885} C_VEL
LIN {X 0,Y 360.942,Z 988.061,A -85,B 0,C 180,E1 6130.009,E2 6130.009} C_VEL
LIN {X 0,Y 371.774,Z 968.65,A -85,B 0,C 180,E1 6129.243,E2 6129.243} C_VEL
LIN {X 0,Y 384.095,Z 943.677,A -85,B 0,C 180,E1 6128.431,E2 6128.431} C_VEL
LIN {X 0,Y 394.092,Z 919.638,A -85,B 0,C 180,E1 6127.803,E2 6127.803} C_VEL
LIN {X 0,Y 401.74,Z 898.293,A -85,B 0,C 180,E1 6127.346,E2 6127.346} C_VEL
LIN {X 0,Y 408.238,Z 876.946,A -85,B 0,C 180,E1 6126.969,E2 6126.969} C_VEL
LIN {X 0,Y 414.37,Z 852.459,A -85,B 0,C 180,E1 6126.626,E2 6126.626} C_VEL
LIN {X 0,Y 419.654,Z 823.659,A -85,B 0,C 180,E1 6126.272,E2 6126.272} C_VEL
LIN {X 0,Y 428.588,Z 751.659,A -85,B 0,C 180,E1 6125.42,E2 6125.42} C_VEL
LIN {X 0,Y 435.59,Z 693.679,A -85,B 0,C 180,E1 6124.707,E2 6124.707} C_VEL
LIN {X 0,Y 435.585,Z 693.81,A -85,B 0,C 180,E1 6122.33,E2 6122.33} C_VEL
LIN {X 0,Y 420.157,Z 820.277,A -85,B 0,C 180,E1 6120.836,E2 6120.836} C_VEL
LIN {X 0,Y 419.028,Z 827.95,A -85,B 0,C 180,E1 6120.894,E2 6120.894} C_VEL
LIN {X 0,Y 414.791,Z 849.426,A -85,B 0,C 180,E1 6121.526,E2 6121.526} C_VEL
LIN {X 0,Y 413.516,Z 854.836,A -85,B 0,C 180,E1 6121.518,E2 6121.518} C_VEL
LIN {X 0,Y 407.596,Z 878.096,A -85,B 0,C 180,E1 6121.222,E2 6121.222} C_VEL
LIN {X 0,Y 401.272,Z 898.664,A -85,B 0,C 180,E1 6120.901,E2 6120.901} C_VEL
LIN {X 0,Y 393.658,Z 919.785,A -85,B 0,C 180,E1 6120.495,E2 6120.495} C_VEL
LIN {X 0,Y 382.945,Z 945.308,A -85,B 0,C 180,E1 6119.889,E2 6119.889} C_VEL
LIN {X 0,Y 370.984,Z 969.268,A -85,B 0,C 180,E1 6119.173,E2 6119.173} C_VEL
LIN {X 0,Y 360.076,Z 988.672,A -85,B 0,C 180,E1 6118.468,E2 6118.468} C_VEL
LIN {X 0,Y 348.736,Z 1006.847,A -85,B 0,C 180,E1 6117.677,E2 6117.677} C_VEL
LIN {X 0,Y 335.511,Z 1026.011,A -85,B 0,C 180,E1 6116.689,E2 6116.689} C_VEL
LIN {X 0,Y 317.571,Z 1049.193,A -85,B 0,C 180,E1 6115.192,E2 6115.192} C_VEL
LIN {X 0,Y 301.963,Z 1067.166,A -85,B 0,C 180,E1 6113.727,E2 6113.727} C_VEL
LIN {X 0,Y 287.45,Z 1082.472,A -85,B 0,C 180,E1 6112.203,E2 6112.203} C_VEL
LIN {X 0,Y 271.801,Z 1097.651,A -85,B 0,C 180,E1 6110.357,E2 6110.357} C_VEL
LIN {X 0,Y 251.836,Z 1115.363,A -85,B 0,C 180,E1 6107.603,E2 6107.603} C_VEL
LIN {X 0,Y 233.385,Z 1130.058,A -85,B 0,C 180,E1 6104.565,E2 6104.565} C_VEL
LIN {X 0,Y 217.324,Z 1141.913,A -85,B 0,C 180,E1 6101.397,E2 6101.397} C_VEL
LIN {X 0,Y 201.207,Z 1153.008,A -85,B 0,C 180,E1 6097.561,E2 6097.561} C_VEL
LIN {X 0,Y 182.348,Z 1165.164,A -85,B 0,C 180,E1 6091.863,E2 6091.863} C_VEL
LIN {X 0,Y 166.366,Z 1174.727,A -85,B 0,C 180,E1 6085.423,E2 6085.423} C_VEL
LIN {X 0,Y 154.134,Z 1181.882,A -85,B 0,C 180,E1 6078.806,E2 6078.806} C_VEL
LIN {X 0,Y 144.017,Z 1187.862,A -85,B 0,C 180,E1 6071.265,E2 6071.265} C_VEL
LIN {X 0,Y 135.705,Z 1193.137,A -85,B 0,C 180,E1 6062.038,E2 6062.038} C_VEL
LIN {X 0,Y 129.91,Z 1197.63,A -85,B 0,C 180,E1 6050.264,E2 6050.264} C_VEL
LIN {X 0,Y 128.124,Z 1199.944,A -85,B 0,C 180,E1 6040.34,E2 6040.34} C_VEL
LIN {X 0,Y 127.916,Z 1201.007,A -85,B 0,C 180,E1 6032.688,E2 6032.688} C_VEL
LIN {X 0,Y 127.915,Z 1201.337,A -85,B 0,C 180,E1 6025.966,E2 6025.966} C_VEL
LIN {X 0,Y 128.297,Z 1201.02,A -85,B 0,C 180,E1 6017.853,E2 6017.853} C_VEL
LIN {X 0,Y 131.094,Z 1199.489,A -85,B 0,C 180,E1 6006.634,E2 6006.634} C_VEL
LIN {X 0,Y 138.153,Z 1196.094,A -85,B 0,C 180,E1 5995.128,E2 5995.128} C_VEL
LIN {X 0,Y 147.528,Z 1191.968,A -85,B 0,C 180,E1 5986.267,E2 5986.267} C_VEL
LIN {X 0,Y 159.1,Z 1186.89,A -85,B 0,C 180,E1 5978.806,E2 5978.806} C_VEL
LIN {X 0,Y 174.155,Z 1180.063,A -85,B 0,C 180,E1 5971.822,E2 5971.822} C_VEL
LIN {X 0,Y 195.06,Z 1169.831,A -85,B 0,C 180,E1 5964.868,E2 5964.868} C_VEL
LIN {X 0,Y 212.433,Z 1160.565,A -85,B 0,C 180,E1 5960.506,E2 5960.506} C_VEL
LIN {X 0,Y 229.125,Z 1150.955,A -85,B 0,C 180,E1 5957.124,E2 5957.124} C_VEL
LIN {X 0,Y 247.677,Z 1139.366,A -85,B 0,C 180,E1 5954.018,E2 5954.018} C_VEL
LIN {X 0,Y 270.833,Z 1123.361,A -85,B 0,C 180,E1 5950.853,E2 5950.853} C_VEL
LIN {X 0,Y 289.415,Z 1109.06,A -85,B 0,C 180,E1 5948.744,E2 5948.744} C_VEL
LIN {X 0,Y 306.297,Z 1094.872,A -85,B 0,C 180,E1 5947.088,E2 5947.088} C_VEL
LIN {X 0,Y 322.538,Z 1079.977,A -85,B 0,C 180,E1 5945.682,E2 5945.682} C_VEL
LIN {X 0,Y 342.165,Z 1060.177,A -85,B 0,C 180,E1 5944.19,E2 5944.19} C_VEL
LIN {X 0,Y 355.085,Z 1045.72,A -85,B 0,C 180,E1 5943.297,E2 5943.297} C_VEL
LIN {X 0,Y 337.164,Z 1065.23,A -85,B 0,C 180,E1 5942.036,E2 5942.036} C_VEL
LIN {X 0,Y 320.981,Z 1081.222,A -85,B 0,C 180,E1 5940.757,E2 5940.757} C_VEL
LIN {X 0,Y 304.977,Z 1095.685,A -85,B 0,C 180,E1 5939.33,E2 5939.33} C_VEL
LIN {X 0,Y 287.225,Z 1110.365,A -85,B 0,C 180,E1 5937.532,E2 5937.532} C_VEL
LIN {X 0,Y 264.062,Z 1127.558,A -85,B 0,C 180,E1 5934.769,E2 5934.769} C_VEL
LIN {X 0,Y 246.233,Z 1139.472,A -85,B 0,C 180,E1 5932.217,E2 5932.217} C_VEL
LIN {X 0,Y 228.964,Z 1150.077,A -85,B 0,C 180,E1 5929.279,E2 5929.279} C_VEL
LIN {X 0,Y 211.53,Z 1159.929,A -85,B 0,C 180,E1 5925.694,E2 5925.694} C_VEL
LIN {X 0,Y 191.09,Z 1170.559,A -85,B 0,C 180,E1 5920.361,E2 5920.361} C_VEL
LIN {X 0,Y 172.57,Z 1179.18,A -85,B 0,C 180,E1 5913.873,E2 5913.873} C_VEL
LIN {X 0,Y 158.979,Z 1185.154,A -85,B 0,C 180,E1 5907.433,E2 5907.433} C_VEL
LIN {X 0,Y 147.369,Z 1190.059,A -85,B 0,C 180,E1 5899.866,E2 5899.866} C_VEL
LIN {X 0,Y 137.193,Z 1194.366,A -85,B 0,C 180,E1 5889.892,E2 5889.892} C_VEL
LIN {X 0,Y 130.508,Z 1197.259,A -85,B 0,C 180,E1 5877.862,E2 5877.862} C_VEL
LIN {X 0,Y 128.395,Z 1198.326,A -85,B 0,C 180,E1 5868.619,E2 5868.619} C_VEL
LIN {X 0,Y 127.936,Z 1198.524,A -85,B 0,C 180,E1 5860.355,E2 5860.355} C_VEL
LIN {X 0,Y 127.925,Z 1198.173,A -85,B 0,C 180,E1 5853.585,E2 5853.585} C_VEL
LIN {X 0,Y 128.324,Z 1197.001,A -85,B 0,C 180,E1 5845.531,E2 5845.531} C_VEL
LIN {X 0,Y 130.936,Z 1194.261,A -85,B 0,C 180,E1 5834.498,E2 5834.498} C_VEL
LIN {X 0,Y 136.903,Z 1190.008,A -85,B 0,C 180,E1 5823.943,E2 5823.943} C_VEL
LIN {X 0,Y 144.88,Z 1185.177,A -85,B 0,C 180,E1 5815.535,E2 5815.535} C_VEL
LIN {X 0,Y 154.803,Z 1179.47,A -85,B 0,C 180,E1 5808.297,E2 5808.297} C_VEL
LIN {X 0,Y 167.27,Z 1172.329,A -85,B 0,C 180,E1 5801.653,E2 5801.653} C_VEL
LIN {X 0,Y 184.909,Z 1161.881,A -85,B 0,C 180,E1 5794.724,E2 5794.724} C_VEL
LIN {X 0,Y 202.337,Z 1150.728,A -85,B 0,C 180,E1 5789.575,E2 5789.575} C_VEL
LIN {X 0,Y 217.851,Z 1140.149,A -85,B 0,C 180,E1 5785.899,E2 5785.899} C_VEL
LIN {X 0,Y 234.095,Z 1128.257,A -85,B 0,C 180,E1 5782.696,E2 5782.696} C_VEL
LIN {X 0,Y 253.524,Z 1112.862,A -85,B 0,C 180,E1 5779.512,E2 5779.512} C_VEL
LIN {X 0,Y 272.697,Z 1095.834,A -85,B 0,C 180,E1 5776.87,E2 5776.87} C_VEL
LIN {X 0,Y 287.853,Z 1081.182,A -85,B 0,C 180,E1 5775.065,E2 5775.065} C_VEL
LIN {X 0,Y 303.255,Z 1064.963,A -85,B 0,C 180,E1 5773.435,E2 5773.435} C_VEL
LIN {X 0,Y 320.999,Z 1044.396,A -85,B 0,C 180,E1 5771.776,E2 5771.776} C_VEL
LIN {X 0,Y 336.558,Z 1023.965,A -85,B 0,C 180,E1 5770.472,E2 5770.472} C_VEL
LIN {X 0,Y 349.247,Z 1005.552,A -85,B 0,C 180,E1 5769.508,E2 5769.508} C_VEL
LIN {X 0,Y 360.439,Z 987.607,A -85,B 0,C 180,E1 5768.706,E2 5768.706} C_VEL
LIN {X 0,Y 372.013,Z 966.964,A -85,B 0,C 180,E1 5767.94,E2 5767.94} C_VEL
LIN {X 0,Y 384.93,Z 940.431,A -85,B 0,C 180,E1 5767.141,E2 5767.141} C_VEL
LIN {X 0,Y 394.059,Z 918.452,A -85,B 0,C 180,E1 5766.606,E2 5766.606} C_VEL
LIN {X 0,Y 401.53,Z 897.637,A -85,B 0,C 180,E1 5766.187,E2 5766.187} C_VEL
LIN {X 0,Y 408.144,Z 875.946,A -85,B 0,C 180,E1 5765.827,E2 5765.827} C_VEL
LIN {X 0,Y 414.893,Z 848.657,A -85,B 0,C 180,E1 5765.472,E2 5765.472} C_VEL
LIN {X 0,Y 419.599,Z 821.991,A -85,B 0,C 180,E1 5765.158,E2 5765.158} C_VEL
LIN {X 0,Y 434.548,Z 701.501,A -85,B 0,C 180,E1 5763.76,E2 5763.76} C_VEL
LIN {X 0,Y 434.523,Z 701.723,A -85,B 0,C 180,E1 5763.296,E2 5763.296} C_VEL
LIN {X 0,Y 419.529,Z 822.57,A -85,B 0,C 180,E1 5761.904,E2 5761.904} C_VEL
LIN {X 0,Y 414.627,Z 850.14,A -85,B 0,C 180,E1 5761.575,E2 5761.575} C_VEL
LIN {X 0,Y 413.516,Z 854.836,A -85,B 0,C 180,E1 5761.518,E2 5761.518} C_VEL
LIN {X 0,Y 411.696,Z 862.372,A -85,B 0,C 180,E1 5761.575,E2 5761.575} C_VEL
LIN {X 0,Y 406.504,Z 881.344,A -85,B 0,C 180,E1 5762.176,E2 5762.176} C_VEL
LIN {X 0,Y 404.276,Z 888.776,A -85,B 0,C 180,E1 5762.202,E2 5762.202} C_VEL
LIN {X 0,Y 395.505,Z 914.045,A -85,B 0,C 180,E1 5761.777,E2 5761.777} C_VEL
LIN {X 0,Y 387.05,Z 934.893,A -85,B 0,C 180,E1 5761.344,E2 5761.344} C_VEL
LIN {X 0,Y 377.987,Z 954.51,A -85,B 0,C 180,E1 5760.853,E2 5760.853} C_VEL
LIN {X 0,Y 367.45,Z 974.743,A -85,B 0,C 180,E1 5760.244,E2 5760.244} C_VEL
LIN {X 0,Y 352.972,Z 999.253,A -85,B 0,C 180,E1 5759.34,E2 5759.34} C_VEL
LIN {X 0,Y 338.589,Z 1020.469,A -85,B 0,C 180,E1 5758.359,E2 5758.359} C_VEL
LIN {X 0,Y 325.206,Z 1038.309,A -85,B 0,C 180,E1 5757.357,E2 5757.357} C_VEL
LIN {X 0,Y 311.37,Z 1055.106,A -85,B 0,C 180,E1 5756.228,E2 5756.228} C_VEL
LIN {X 0,Y 293.277,Z 1075.102,A -85,B 0,C 180,E1 5754.562,E2 5754.562} C_VEL
LIN {X 0,Y 274.272,Z 1093.679,A -85,B 0,C 180,E1 5752.555,E2 5752.555} C_VEL
LIN {X 0,Y 258.419,Z 1107.864,A -85,B 0,C 180,E1 5750.619,E2 5750.619} C_VEL
LIN {X 0,Y 241.991,Z 1121.402,A -85,B 0,C 180,E1 5748.303,E2 5748.303} C_VEL
LIN {X 0,Y 222.515,Z 1136.177,A -85,B 0,C 180,E1 5745.036,E2 5745.036} C_VEL
LIN {X 0,Y 202.205,Z 1150.019,A -85,B 0,C 180,E1 5740.812,E2 5740.812} C_VEL
LIN {X 0,Y 185.914,Z 1160.315,A -85,B 0,C 180,E1 5736.547,E2 5736.547} C_VEL
LIN {X 0,Y 170.649,Z 1169.387,A -85,B 0,C 180,E1 5731.506,E2 5731.506} C_VEL
LIN {X 0,Y 154.066,Z 1178.823,A -85,B 0,C 180,E1 5724.215,E2 5724.215} C_VEL
LIN {X 0,Y 139.731,Z 1186.607,A -85,B 0,C 180,E1 5715.105,E2 5715.105} C_VEL
LIN {X 0,Y 130.804,Z 1191.677,A -85,B 0,C 180,E1 5706.6,E2 5706.6} C_VEL
LIN {X 0,Y 124.792,Z 1195.481,A -85,B 0,C 180,E1 5697.691,E2 5697.691} C_VEL
LIN {X 0,Y 121.415,Z 1198.192,A -85,B 0,C 180,E1 5688.726,E2 5688.726} C_VEL
LIN {X 0,Y 120.103,Z 1199.964,A -85,B 0,C 180,E1 5680.068,E2 5680.068} C_VEL
LIN {X 0,Y 119.917,Z 1200.932,A -85,B 0,C 180,E1 5672.389,E2 5672.389} C_VEL
LIN {X 0,Y 119.922,Z 1201.26,A -85,B 0,C 180,E1 5665.217,E2 5665.217} C_VEL
LIN {X 0,Y 120.5,Z 1200.891,A -85,B 0,C 180,E1 5656.076,E2 5656.076} C_VEL
LIN {X 0,Y 124.005,Z 1199.234,A -85,B 0,C 180,E1 5644.189,E2 5644.189} C_VEL
LIN {X 0,Y 131.803,Z 1195.916,A -85,B 0,C 180,E1 5632.636,E2 5632.636} C_VEL
LIN {X 0,Y 141.61,Z 1191.973,A -85,B 0,C 180,E1 5623.93,E2 5623.93} C_VEL
LIN {X 0,Y 153.99,Z 1186.917,A -85,B 0,C 180,E1 5616.377,E2 5616.377} C_VEL
LIN {X 0,Y 169.177,Z 1180.419,A -85,B 0,C 180,E1 5609.682,E2 5609.682} C_VEL
LIN {X 0,Y 190.893,Z 1170.335,A -85,B 0,C 180,E1 5602.802,E2 5602.802} C_VEL
LIN {X 0,Y 209.771,Z 1160.626,A -85,B 0,C 180,E1 5598.336,E2 5598.336} C_VEL
LIN {X 0,Y 227.679,Z 1150.602,A -85,B 0,C 180,E1 5594.954,E2 5594.954} C_VEL
LIN {X 0,Y 247.519,Z 1138.476,A -85,B 0,C 180,E1 5591.889,E2 5591.889} C_VEL
LIN {X 0,Y 271.236,Z 1122.254,A -85,B 0,C 180,E1 5588.913,E2 5588.913} C_VEL
LIN {X 0,Y 289.136,Z 1108.66,A -85,B 0,C 180,E1 5587.037,E2 5587.037} C_VEL
LIN {X 0,Y 306.353,Z 1094.363,A -85,B 0,C 180,E1 5585.474,E2 5585.474} C_VEL
LIN {X 0,Y 322.804,Z 1079.426,A -85,B 0,C 180,E1 5584.16,E2 5584.16} C_VEL
LIN {X 0,Y 334.734,Z 1067.667,A -85,B 0,C 180,E1 5583.284,E2 5583.284} C_VEL
LIN {X 0,Y 318.665,Z 1083.2,A -85,B 0,C 180,E1 5582.086,E2 5582.086} C_VEL
LIN {X 0,Y 298.724,Z 1100.73,A -85,B 0,C 180,E1 5580.384,E2 5580.384} C_VEL
LIN {X 0,Y 277.092,Z 1117.53,A -85,B 0,C 180,E1 5578.23,E2 5578.23} C_VEL
LIN {X 0,Y 259.541,Z 1129.911,A -85,B 0,C 180,E1 5576.173,E2 5576.173} C_VEL
LIN {X 0,Y 242.373,Z 1141.012,A -85,B 0,C 180,E1 5573.822,E2 5573.822} C_VEL
LIN {X 0,Y 223.848,Z 1151.991,A -85,B 0,C 180,E1 5570.799,E2 5570.799} C_VEL
LIN {X 0,Y 200.867,Z 1164.276,A -85,B 0,C 180,E1 5566.084,E2 5566.084} C_VEL
LIN {X 0,Y 182.299,Z 1173.148,A -85,B 0,C 180,E1 5561.119,E2 5561.119} C_VEL
LIN {X 0,Y 166.745,Z 1180.019,A -85,B 0,C 180,E1 5555.705,E2 5555.705} C_VEL
LIN {X 0,Y 152.547,Z 1185.878,A -85,B 0,C 180,E1 5549.163,E2 5549.163} C_VEL
LIN {X 0,Y 138.026,Z 1191.636,A -85,B 0,C 180,E1 5539.518,E2 5539.518} C_VEL
LIN {X 0,Y 127.6,Z 1195.509,A -85,B 0,C 180,E1 5528.245,E2 5528.245} C_VEL
LIN {X 0,Y 122.525,Z 1197.521,A -85,B 0,C 180,E1 5518.193,E2 5518.193} C_VEL
LIN {X 0,Y 120.405,Z 1198.451,A -85,B 0,C 180,E1 5508.789,E2 5508.789} C_VEL
LIN {X 0,Y 119.936,Z 1198.589,A -85,B 0,C 180,E1 5500.341,E2 5500.341} C_VEL
LIN {X 0,Y 119.932,Z 1198.201,A -85,B 0,C 180,E1 5492.867,E2 5492.867} C_VEL
LIN {X 0,Y 120.517,Z 1196.924,A -85,B 0,C 180,E1 5483.809,E2 5483.809} C_VEL
LIN {X 0,Y 123.782,Z 1193.963,A -85,B 0,C 180,E1 5472.125,E2 5472.125} C_VEL
LIN {X 0,Y 129.976,Z 1190.033,A -85,B 0,C 180,E1 5462.015,E2 5462.015} C_VEL
LIN {X 0,Y 138.731,Z 1185.151,A -85,B 0,C 180,E1 5453.26,E2 5453.26} C_VEL
LIN {X 0,Y 149.953,Z 1179.126,A -85,B 0,C 180,E1 5445.564,E2 5445.564} C_VEL
LIN {X 0,Y 165.211,Z 1170.878,A -85,B 0,C 180,E1 5438.117,E2 5438.117} C_VEL
LIN {X 0,Y 184.048,Z 1159.966,A -85,B 0,C 180,E1 5431.47,E2 5431.47} C_VEL
LIN {X 0,Y 200.01,Z 1150.075,A -85,B 0,C 180,E1 5427.149,E2 5427.149} C_VEL
LIN {X 0,Y 216.063,Z 1139.41,A -85,B 0,C 180,E1 5423.614,E2 5423.614} C_VEL
LIN {X 0,Y 235.351,Z 1125.559,A -85,B 0,C 180,E1 5420.129,E2 5420.129} C_VEL
LIN {X 0,Y 255.318,Z 1109.578,A -85,B 0,C 180,E1 5417.151,E2 5417.151} C_VEL
LIN {X 0,Y 272.26,Z 1094.698,A -85,B 0,C 180,E1 5415.018,E2 5415.018} C_VEL
LIN {X 0,Y 287.694,Z 1079.927,A -85,B 0,C 180,E1 5413.316,E2 5413.316} C_VEL
LIN {X 0,Y 304.738,Z 1062.086,A -85,B 0,C 180,E1 5411.654,E2 5411.654} C_VEL
LIN {X 0,Y 322.941,Z 1040.659,A -85,B 0,C 180,E1 5410.083,E2 5410.083} C_VEL
LIN {X 0,Y 336.615,Z 1022.744,A -85,B 0,C 180,E1 5409.021,E2 5409.021} C_VEL
LIN {X 0,Y 348.971,Z 1004.918,A -85,B 0,C 180,E1 5408.147,E2 5408.147} C_VEL
LIN {X 0,Y 360.913,Z 985.841,A -85,B 0,C 180,E1 5407.349,E2 5407.349} C_VEL
LIN {X 0,Y 374.372,Z 961.654,A -85,B 0,C 180,E1 5406.527,E2 5406.527} C_VEL
LIN {X 0,Y 385.477,Z 938.291,A -85,B 0,C 180,E1 5405.887,E2 5405.887} C_VEL
LIN {X 0,Y 394.198,Z 917.266,A -85,B 0,C 180,E1 5405.409,E2 5405.409} C_VEL
LIN {X 0,Y 401.83,Z 895.956,A -85,B 0,C 180,E1 5405.01,E2 5405.01} C_VEL
LIN {X 0,Y 409.389,Z 870.836,A -85,B 0,C 180,E1 5404.63,E2 5404.63} C_VEL
LIN {X 0,Y 415.797,Z 843.007,A -85,B 0,C 180,E1 5404.3,E2 5404.3} C_VEL
LIN {X 0,Y 419.717,Z 820.226,A -85,B 0,C 180,E1 5404.042,E2 5404.042} C_VEL
LIN {X 0,Y 425.441,Z 775.48,A -85,B 0,C 180,E1 5403.53,E2 5403.53} C_VEL
LIN {X 0,Y 418.824,Z 826.395,A -85,B 0,C 180,E1 5402.956,E2 5402.956} C_VEL
LIN {X 0,Y 413.122,Z 855.612,A -85,B 0,C 180,E1 5402.621,E2 5402.621} C_VEL
LIN {X 0,Y 407.282,Z 878.304,A -85,B 0,C 180,E1 5402.347,E2 5402.347} C_VEL
LIN {X 0,Y 404.276,Z 888.776,A -85,B 0,C 180,E1 5402.202,E2 5402.202} C_VEL
LIN {X 0,Y 401.906,Z 896.169,A -85,B 0,C 180,E1 5402.233,E2 5402.233} C_VEL
LIN {X 0,Y 395.075,Z 914.727,A -85,B 0,C 180,E1 5402.79,E2 5402.79} C_VEL
LIN {X 0,Y 392.267,Z 921.929,A -85,B 0,C 180,E1 5402.799,E2 5402.799} C_VEL
LIN {X 0,Y 380.226,Z 949.32,A -85,B 0,C 180,E1 5402.206,E2 5402.206} C_VEL
LIN {X 0,Y 369.599,Z 970.077,A -85,B 0,C 180,E1 5401.647,E2 5401.647} C_VEL
LIN {X 0,Y 358.684,Z 989.084,A -85,B 0,C 180,E1 5401.031,E2 5401.031} C_VEL
LIN {X 0,Y 346.955,Z 1007.468,A -85,B 0,C 180,E1 5400.318,E2 5400.318} C_VEL
LIN {X 0,Y 331.664,Z 1029.037,A -85,B 0,C 180,E1 5399.309,E2 5399.309} C_VEL
LIN {X 0,Y 314.142,Z 1050.753,A -85,B 0,C 180,E1 5398.02,E2 5398.02} C_VEL
LIN {X 0,Y 299.422,Z 1067.231,A -85,B 0,C 180,E1 5396.803,E2 5396.803} C_VEL
LIN {X 0,Y 284.365,Z 1082.65,A -85,B 0,C 180,E1 5395.423,E2 5395.423} C_VEL
LIN {X 0,Y 267.586,Z 1098.38,A -85,B 0,C 180,E1 5393.682,E2 5393.682} C_VEL
LIN {X 0,Y 245.966,Z 1116.654,A -85,B 0,C 180,E1 5391.039,E2 5391.039} C_VEL
LIN {X 0,Y 227.652,Z 1130.558,A -85,B 0,C 180,E1 5388.356,E2 5388.356} C_VEL
LIN {X 0,Y 210.778,Z 1142.346,A -85,B 0,C 180,E1 5385.398,E2 5385.398} C_VEL
LIN {X 0,Y 192.824,Z 1153.934,A -85,B 0,C 180,E1 5381.56,E2 5381.56} C_VEL
LIN {X 0,Y 171.295,Z 1166.599,A -85,B 0,C 180,E1 5375.585,E2 5375.585} C_VEL
LIN {X 0,Y 156.008,Z 1174.933,A -85,B 0,C 180,E1 5369.907,E2 5369.907} C_VEL
LIN {X 0,Y 142.405,Z 1182.036,A -85,B 0,C 180,E1 5363.17,E2 5363.17} C_VEL
LIN {X 0,Y 130.416,Z 1188.226,A -85,B 0,C 180,E1 5354.856,E2 5354.856} C_VEL
LIN {X 0,Y 119.581,Z 1194.166,A -85,B 0,C 180,E1 5342.921,E2 5342.921} C_VEL
LIN {X 0,Y 113.995,Z 1197.815,A -85,B 0,C 180,E1 5331.076,E2 5331.076} C_VEL
LIN {X 0,Y 112.147,Z 1199.845,A -85,B 0,C 180,E1 5320.791,E2 5320.791} C_VEL
LIN {X 0,Y 111.916,Z 1200.834,A -85,B 0,C 180,E1 5312.56,E2 5312.56} C_VEL
LIN {X 0,Y 111.92,Z 1201.141,A -85,B 0,C 180,E1 5305.388,E2 5305.388} C_VEL
LIN {X 0,Y 112.478,Z 1200.862,A -85,B 0,C 180,E1 5296.113,E2 5296.113} C_VEL
LIN {X 0,Y 115.944,Z 1199.443,A -85,B 0,C 180,E1 5283.908,E2 5283.908} C_VEL
LIN {X 0,Y 124.882,Z 1196.061,A -85,B 0,C 180,E1 5270.765,E2 5270.765} C_VEL
LIN {X 0,Y 135.947,Z 1191.979,A -85,B 0,C 180,E1 5261.394,E2 5261.394} C_VEL
LIN {X 0,Y 149.169,Z 1186.948,A -85,B 0,C 180,E1 5253.783,E2 5253.783} C_VEL
LIN {X 0,Y 165.186,Z 1180.473,A -85,B 0,C 180,E1 5247.155,E2 5247.155} C_VEL
LIN {X 0,Y 186.986,Z 1170.84,A -85,B 0,C 180,E1 5240.648,E2 5240.648} C_VEL
LIN {X 0,Y 207.162,Z 1160.823,A -85,B 0,C 180,E1 5236.166,E2 5236.166} C_VEL
LIN {X 0,Y 225.668,Z 1150.763,A -85,B 0,C 180,E1 5232.905,E2 5232.905} C_VEL
LIN {X 0,Y 245.077,Z 1139.195,A -85,B 0,C 180,E1 5230.104,E2 5230.104} C_VEL
LIN {X 0,Y 269.397,Z 1123.004,A -85,B 0,C 180,E1 5227.25,E2 5227.25} C_VEL
LIN {X 0,Y 288.736,Z 1108.558,A -85,B 0,C 180,E1 5225.365,E2 5225.365} C_VEL
LIN {X 0,Y 305.701,Z 1094.666,A -85,B 0,C 180,E1 5223.939,E2 5223.939} C_VEL
LIN {X 0,Y 314.255,Z 1087.27,A -85,B 0,C 180,E1 5223.26,E2 5223.26} C_VEL
LIN {X 0,Y 293.063,Z 1105.01,A -85,B 0,C 180,E1 5221.534,E2 5221.534} C_VEL
LIN {X 0,Y 274.696,Z 1118.876,A -85,B 0,C 180,E1 5219.791,E2 5219.791} C_VEL
LIN {X 0,Y 257.142,Z 1130.966,A -85,B 0,C 180,E1 5217.859,E2 5217.859} C_VEL
LIN {X 0,Y 237.751,Z 1143.143,A -85,B 0,C 180,E1 5215.342,E2 5215.342} C_VEL
LIN {X 0,Y 213.088,Z 1156.947,A -85,B 0,C 180,E1 5211.364,E2 5211.364} C_VEL
LIN {X 0,Y 194.415,Z 1166.271,A -85,B 0,C 180,E1 5207.525,E2 5207.525} C_VEL
LIN {X 0,Y 177.58,Z 1173.951,A -85,B 0,C 180,E1 5203.172,E2 5203.172} C_VEL
LIN {X 0,Y 161.073,Z 1180.87,A -85,B 0,C 180,E1 5197.655,E2 5197.655} C_VEL
LIN {X 0,Y 143.043,Z 1187.872,A -85,B 0,C 180,E1 5189.289,E2 5189.289} C_VEL
LIN {X 0,Y 128.508,Z 1192.936,A -85,B 0,C 180,E1 5179,E2 5179} C_VEL
LIN {X 0,Y 119.946,Z 1195.879,A -85,B 0,C 180,E1 5169.311,E2 5169.311} C_VEL
LIN {X 0,Y 114.77,Z 1197.702,A -85,B 0,C 180,E1 5159.2,E2 5159.2} C_VEL
LIN {X 0,Y 112.488,Z 1198.552,A -85,B 0,C 180,E1 5149.571,E2 5149.571} C_VEL
LIN {X 0,Y 111.939,Z 1198.673,A -85,B 0,C 180,E1 5140.711,E2 5140.711} C_VEL
LIN {X 0,Y 111.929,Z 1198.319,A -85,B 0,C 180,E1 5133.072,E2 5133.072} C_VEL
LIN {X 0,Y 112.492,Z 1197.114,A -85,B 0,C 180,E1 5123.877,E2 5123.877} C_VEL
LIN {X 0,Y 115.935,Z 1194.292,A -85,B 0,C 180,E1 5111.392,E2 5111.392} C_VEL
LIN {X 0,Y 122.9,Z 1190.23,A -85,B 0,C 180,E1 5100.247,E2 5100.247} C_VEL
LIN {X 0,Y 132.325,Z 1185.372,A -85,B 0,C 180,E1 5091.16,E2 5091.16} C_VEL
LIN {X 0,Y 144.147,Z 1179.433,A -85,B 0,C 180,E1 5083.372,E2 5083.372} C_VEL
LIN {X 0,Y 158.951,Z 1171.842,A -85,B 0,C 180,E1 5076.374,E2 5076.374} C_VEL
LIN {X 0,Y 179.174,Z 1160.739,A -85,B 0,C 180,E1 5069.479,E2 5069.479} C_VEL
LIN {X 0,Y 196.432,Z 1150.428,A -85,B 0,C 180,E1 5065.037,E2 5065.037} C_VEL
LIN {X 0,Y 212.938,Z 1139.792,A -85,B 0,C 180,E1 5061.61,E2 5061.61} C_VEL
LIN {X 0,Y 230.932,Z 1127.22,A -85,B 0,C 180,E1 5058.524,E2 5058.524} C_VEL
LIN {X 0,Y 253.049,Z 1110.06,A -85,B 0,C 180,E1 5055.399,E2 5055.399} C_VEL
LIN {X 0,Y 270.28,Z 1095.217,A -85,B 0,C 180,E1 5053.364,E2 5053.364} C_VEL
LIN {X 0,Y 285.946,Z 1080.479,A -85,B 0,C 180,E1 5051.745,E2 5051.745} C_VEL
LIN {X 0,Y 301.806,Z 1064.164,A -85,B 0,C 180,E1 5050.285,E2 5050.285} C_VEL
LIN {X 0,Y 321.161,Z 1041.94,A -85,B 0,C 180,E1 5048.714,E2 5048.714} C_VEL
LIN {X 0,Y 335.933,Z 1022.831,A -85,B 0,C 180,E1 5047.639,E2 5047.639} C_VEL
LIN {X 0,Y 348.411,Z 1005.003,A -85,B 0,C 180,E1 5046.815,E2 5046.815} C_VEL
LIN {X 0,Y 360.465,Z 985.923,A -85,B 0,C 180,E1 5046.064,E2 5046.064} C_VEL
LIN {X 0,Y 374.039,Z 961.733,A -85,B 0,C 180,E1 5045.29,E2 5045.29} C_VEL
LIN {X 0,Y 385.233,Z 938.367,A -85,B 0,C 180,E1 5044.689,E2 5044.689} C_VEL
LIN {X 0,Y 394.021,Z 917.338,A -85,B 0,C 180,E1 5044.239,E2 5044.239} C_VEL
LIN {X 0,Y 401.606,Z 896.324,A -85,B 0,C 180,E1 5043.868,E2 5043.868} C_VEL
LIN {X 0,Y 408.561,Z 873.528,A -85,B 0,C 180,E1 5043.534,E2 5043.534} C_VEL
LIN {X 0,Y 401.579,Z 896.437,A -85,B 0,C 180,E1 5043.229,E2 5043.229} C_VEL
LIN {X 0,Y 394.194,Z 916.955,A -85,B 0,C 180,E1 5042.891,E2 5042.891} C_VEL
LIN {X 0,Y 392.267,Z 921.929,A -85,B 0,C 180,E1 5042.799,E2 5042.799} C_VEL
LIN {X 0,Y 389.344,Z 929.148,A -85,B 0,C 180,E1 5042.804,E2 5042.804} C_VEL
LIN {X 0,Y 380.647,Z 948.263,A -85,B 0,C 180,E1 5043.333,E2 5043.333} C_VEL
LIN {X 0,Y 377.714,Z 954.123,A -85,B 0,C 180,E1 5043.311,E2 5043.311} C_VEL
LIN {X 0,Y 366.876,Z 974.629,A -85,B 0,C 180,E1 5042.772,E2 5042.772} C_VEL
LIN {X 0,Y 352.159,Z 999.124,A -85,B 0,C 180,E1 5041.979,E2 5041.979} C_VEL
LIN {X 0,Y 337.34,Z 1020.569,A -85,B 0,C 180,E1 5041.104,E2 5041.104} C_VEL
LIN {X 0,Y 323.955,Z 1038.048,A -85,B 0,C 180,E1 5040.242,E2 5040.242} C_VEL
LIN {X 0,Y 309.483,Z 1055.23,A -85,B 0,C 180,E1 5039.219,E2 5039.219} C_VEL
LIN {X 0,Y 290.688,Z 1075.444,A -85,B 0,C 180,E1 5037.716,E2 5037.716} C_VEL
LIN {X 0,Y 271.632,Z 1093.528,A -85,B 0,C 180,E1 5035.969,E2 5035.969} C_VEL
LIN {X 0,Y 255.255,Z 1107.717,A -85,B 0,C 180,E1 5034.231,E2 5034.231} C_VEL
LIN {X 0,Y 239.139,Z 1120.536,A -85,B 0,C 180,E1 5032.268,E2 5032.268} C_VEL
LIN {X 0,Y 221.501,Z 1133.417,A -85,B 0,C 180,E1 5029.753,E2 5029.753} C_VEL
LIN {X 0,Y 199.049,Z 1148.275,A -85,B 0,C 180,E1 5025.805,E2 5025.805} C_VEL
LIN {X 0,Y 180.016,Z 1159.589,A -85,B 0,C 180,E1 5021.542,E2 5021.542} C_VEL
LIN {X 0,Y 164.034,Z 1168.392,A -85,B 0,C 180,E1 5016.986,E2 5016.986} C_VEL
LIN {X 0,Y 148.36,Z 1176.486,A -85,B 0,C 180,E1 5011.177,E2 5011.177} C_VEL
LIN {X 0,Y 131.35,Z 1184.875,A -85,B 0,C 180,E1 5002.341,E2 5002.341} C_VEL
LIN {X 0,Y 118.281,Z 1191.089,A -85,B 0,C 180,E1 4991.898,E2 4991.898} C_VEL
LIN {X 0,Y 110.393,Z 1195.168,A -85,B 0,C 180,E1 4981.635,E2 4981.635} C_VEL
LIN {X 0,Y 105.889,Z 1198.024,A -85,B 0,C 180,E1 4971.027,E2 4971.027} C_VEL
LIN {X 0,Y 104.161,Z 1199.796,A -85,B 0,C 180,E1 4961.068,E2 4961.068} C_VEL
LIN {X 0,Y 103.917,Z 1200.759,A -85,B 0,C 180,E1 4952.206,E2 4952.206} C_VEL
LIN {X 0,Y 103.932,Z 1201.064,A -85,B 0,C 180,E1 4944.479,E2 4944.479} C_VEL
LIN {X 0,Y 104.786,Z 1200.734,A -85,B 0,C 180,E1 4933.936,E2 4933.936} C_VEL
LIN {X 0,Y 109.598,Z 1199.08,A -85,B 0,C 180,E1 4920.079,E2 4920.079} C_VEL
LIN {X 0,Y 119.469,Z 1195.723,A -85,B 0,C 180,E1 4907.32,E2 4907.32} C_VEL
LIN {X 0,Y 131.162,Z 1191.78,A -85,B 0,C 180,E1 4898.263,E2 4898.263} C_VEL
LIN {X 0,Y 145.364,Z 1186.726,A -85,B 0,C 180,E1 4890.708,E2 4890.708} C_VEL
LIN {X 0,Y 162.309,Z 1180.226,A -85,B 0,C 180,E1 4884.257,E2 4884.257} C_VEL
LIN {X 0,Y 185.885,Z 1170.141,A -85,B 0,C 180,E1 4877.812,E2 4877.812} C_VEL
LIN {X 0,Y 205.88,Z 1160.502,A -85,B 0,C 180,E1 4873.76,E2 4873.76} C_VEL
LIN {X 0,Y 224.107,Z 1150.84,A -85,B 0,C 180,E1 4870.801,E2 4870.801} C_VEL
LIN {X 0,Y 243.462,Z 1139.564,A -85,B 0,C 180,E1 4868.213,E2 4868.213} C_VEL
LIN {X 0,Y 267.245,Z 1124.142,A -85,B 0,C 180,E1 4865.619,E2 4865.619} C_VEL
LIN {X 0,Y 287.582,Z 1109.234,A -85,B 0,C 180,E1 4863.774,E2 4863.774} C_VEL
LIN {X 0,Y 293.89,Z 1104.336,A -85,B 0,C 180,E1 4863.254,E2 4863.254} C_VEL
LIN {X 0,Y 275.07,Z 1118.41,A -85,B 0,C 180,E1 4861.619,E2 4861.619} C_VEL
LIN {X 0,Y 256.821,Z 1130.817,A -85,B 0,C 180,E1 4859.777,E2 4859.777} C_VEL
LIN {X 0,Y 238.18,Z 1142.347,A -85,B 0,C 180,E1 4857.567,E2 4857.567} C_VEL
LIN {X 0,Y 215.066,Z 1155.255,A -85,B 0,C 180,E1 4854.21,E2 4854.21} C_VEL
LIN {X 0,Y 192.846,Z 1166.082,A -85,B 0,C 180,E1 4850.097,E2 4850.097} C_VEL
LIN {X 0,Y 175.242,Z 1173.852,A -85,B 0,C 180,E1 4845.918,E2 4845.918} C_VEL
LIN {X 0,Y 157.951,Z 1180.798,A -85,B 0,C 180,E1 4840.595,E2 4840.595} C_VEL
LIN {X 0,Y 138.791,Z 1187.843,A -85,B 0,C 180,E1 4832.387,E2 4832.387} C_VEL
LIN {X 0,Y 122.999,Z 1192.942,A -85,B 0,C 180,E1 4822.046,E2 4822.046} C_VEL
LIN {X 0,Y 113.441,Z 1195.91,A -85,B 0,C 180,E1 4812.056,E2 4812.056} C_VEL
LIN {X 0,Y 107.461,Z 1197.758,A -85,B 0,C 180,E1 4801.403,E2 4801.403} C_VEL
LIN {X 0,Y 104.62,Z 1198.645,A -85,B 0,C 180,E1 4790.708,E2 4790.708} C_VEL
LIN {X 0,Y 103.951,Z 1198.778,A -85,B 0,C 180,E1 4781.653,E2 4781.653} C_VEL
LIN {X 0,Y 103.923,Z 1198.449,A -85,B 0,C 180,E1 4773.862,E2 4773.862} C_VEL
LIN {X 0,Y 104.403,Z 1197.37,A -85,B 0,C 180,E1 4764.505,E2 4764.505} C_VEL
LIN {X 0,Y 107.669,Z 1194.902,A -85,B 0,C 180,E1 4751.595,E2 4751.595} C_VEL
LIN {X 0,Y 115.562,Z 1190.628,A -85,B 0,C 180,E1 4738.726,E2 4738.726} C_VEL
LIN {X 0,Y 126.114,Z 1185.594,A -85,B 0,C 180,E1 4728.85,E2 4728.85} C_VEL
LIN {X 0,Y 138.31,Z 1179.862,A -85,B 0,C 180,E1 4721.138,E2 4721.138} C_VEL
LIN {X 0,Y 152.85,Z 1172.802,A -85,B 0,C 180,E1 4714.491,E2 4714.491} C_VEL
LIN {X 0,Y 172.185,Z 1162.853,A -85,B 0,C 180,E1 4708.038,E2 4708.038} C_VEL
LIN {X 0,Y 192.301,Z 1151.284,A -85,B 0,C 180,E1 4703.03,E2 4703.03} C_VEL
LIN {X 0,Y 209.22,Z 1140.735,A -85,B 0,C 180,E1 4699.702,E2 4699.702} C_VEL
LIN {X 0,Y 226.708,Z 1128.876,A -85,B 0,C 180,E1 4696.856,E2 4696.856} C_VEL
LIN {X 0,Y 247.381,Z 1113.532,A -85,B 0,C 180,E1 4694.065,E2 4694.065} C_VEL
LIN {X 0,Y 267.601,Z 1096.554,A -85,B 0,C 180,E1 4691.783,E2 4691.783} C_VEL
LIN {X 0,Y 283.475,Z 1081.932,A -85,B 0,C 180,E1 4690.241,E2 4690.241} C_VEL
LIN {X 0,Y 298.575,Z 1066.739,A -85,B 0,C 180,E1 4688.929,E2 4688.929} C_VEL
LIN {X 0,Y 314.294,Z 1049.399,A -85,B 0,C 180,E1 4687.708,E2 4687.708} C_VEL
LIN {X 0,Y 333.034,Z 1026.191,A -85,B 0,C 180,E1 4686.411,E2 4686.411} C_VEL
LIN {X 0,Y 346.894,Z 1006.791,A -85,B 0,C 180,E1 4685.55,E2 4685.55} C_VEL
LIN {X 0,Y 358.736,Z 988.395,A -85,B 0,C 180,E1 4684.858,E2 4684.858} C_VEL
LIN {X 0,Y 369.964,Z 968.973,A -85,B 0,C 180,E1 4684.252,E2 4684.252} C_VEL
LIN {X 0,Y 382.214,Z 945.05,A -85,B 0,C 180,E1 4683.636,E2 4683.636} C_VEL
LIN {X 0,Y 383.362,Z 942.499,A -85,B 0,C 180,E1 4683.579,E2 4683.579} C_VEL
LIN {X 0,Y 377.714,Z 954.123,A -85,B 0,C 180,E1 4683.311,E2 4683.311} C_VEL
LIN {X 0,Y 377.499,Z 955.045,A -85,B 0,C 180,E1 4683.301,E2 4683.301} C_VEL
LIN {X 0,Y 377.499,Z 1003.078,A -85,B 0,C 180,E1 4683.301,E2 4683.301} C_VEL
LIN {X 0,Y 363.335,Z 1003.078,A -85,B 0,C 180,E1 4683.714,E2 4683.714} C_VEL
LIN {X 0,Y 361.371,Z 1001.078,A -85,B 0,C 180,E1 4683.773,E2 4683.773} C_VEL
LIN {X 0,Y 361.371,Z 990.84,A -85,B 0,C 180,E1 4683.773,E2 4683.773} C_VEL
LIN {X 0,Y 357.852,Z 989.757,A -85,B 0,C 180,E1 4683.601,E2 4683.601} C_VEL
LIN {X 0,Y 345.408,Z 1008.842,A -85,B 0,C 180,E1 4682.951,E2 4682.951} C_VEL
LIN {X 0,Y 328.145,Z 1032.364,A -85,B 0,C 180,E1 4681.967,E2 4681.967} C_VEL
LIN {X 0,Y 311.733,Z 1052.039,A -85,B 0,C 180,E1 4680.919,E2 4680.919} C_VEL
LIN {X 0,Y 296.957,Z 1068.116,A -85,B 0,C 180,E1 4679.865,E2 4679.865} C_VEL
LIN {X 0,Y 281.042,Z 1083.915,A -85,B 0,C 180,E1 4678.606,E2 4678.606} C_VEL
LIN {X 0,Y 260.39,Z 1102.493,A -85,B 0,C 180,E1 4676.714,E2 4676.714} C_VEL
LIN {X 0,Y 239.932,Z 1118.754,A -85,B 0,C 180,E1 4674.5,E2 4674.5} C_VEL
LIN {X 0,Y 222.434,Z 1131.426,A -85,B 0,C 180,E1 4672.25,E2 4672.25} C_VEL
LIN {X 0,Y 204.409,Z 1143.369,A -85,B 0,C 180,E1 4669.477,E2 4669.477} C_VEL
LIN {X 0,Y 182.049,Z 1156.811,A -85,B 0,C 180,E1 4665.157,E2 4665.157} C_VEL
LIN {X 0,Y 162.493,Z 1167.3,A -85,B 0,C 180,E1 4660.218,E2 4660.218} C_VEL
LIN {X 0,Y 146.736,Z 1175.132,A -85,B 0,C 180,E1 4654.993,E2 4654.993} C_VEL
LIN {X 0,Y 131.643,Z 1182.184,A -85,B 0,C 180,E1 4648.284,E2 4648.284} C_VEL
LIN {X 0,Y 116.83,Z 1188.879,A -85,B 0,C 180,E1 4638.776,E2 4638.776} C_VEL
LIN {X 0,Y 104.393,Z 1194.556,A -85,B 0,C 180,E1 4625.497,E2 4625.497} C_VEL
LIN {X 0,Y 98.47,Z 1197.766,A -85,B 0,C 180,E1 4613.328,E2 4613.328} C_VEL
LIN {X 0,Y 96.229,Z 1199.677,A -85,B 0,C 180,E1 4601.994,E2 4601.994} C_VEL
LIN {X 0,Y 95.916,Z 1200.661,A -85,B 0,C 180,E1 4592.39,E2 4592.39} C_VEL
LIN {X 0,Y 95.94,Z 1200.966,A -85,B 0,C 180,E1 4584.018,E2 4584.018} C_VEL
LIN {X 0,Y 96.989,Z 1200.655,A -85,B 0,C 180,E1 4572.605,E2 4572.605} C_VEL
LIN {X 0,Y 102.317,Z 1199.111,A -85,B 0,C 180,E1 4558.15,E2 4558.15} C_VEL
LIN {X 0,Y 113.493,Z 1195.708,A -85,B 0,C 180,E1 4544.472,E2 4544.472} C_VEL
LIN {X 0,Y 126.796,Z 1191.581,A -85,B 0,C 180,E1 4534.905,E2 4534.905} C_VEL
LIN {X 0,Y 142.004,Z 1186.503,A -85,B 0,C 180,E1 4527.48,E2 4527.48} C_VEL
LIN {X 0,Y 160.664,Z 1179.677,A -85,B 0,C 180,E1 4521.014,E2 4521.014} C_VEL
LIN {X 0,Y 185.25,Z 1169.446,A -85,B 0,C 180,E1 4514.956,E2 4514.956} C_VEL
LIN {X 0,Y 204.966,Z 1160.185,A -85,B 0,C 180,E1 4511.332,E2 4511.332} C_VEL
LIN {X 0,Y 223.474,Z 1150.582,A -85,B 0,C 180,E1 4508.588,E2 4508.588} C_VEL
LIN {X 0,Y 243.742,Z 1138.971,A -85,B 0,C 180,E1 4506.123,E2 4506.123} C_VEL
LIN {X 0,Y 269.117,Z 1122.588,A -85,B 0,C 180,E1 4503.621,E2 4503.621} C_VEL
LIN {X 0,Y 273.398,Z 1119.566,A -85,B 0,C 180,E1 4503.241,E2 4503.241} C_VEL
LIN {X 0,Y 255.053,Z 1131.779,A -85,B 0,C 180,E1 4501.524,E2 4501.524} C_VEL
LIN {X 0,Y 232.626,Z 1145.282,A -85,B 0,C 180,E1 4499.015,E2 4499.015} C_VEL
LIN {X 0,Y 208.57,Z 1157.908,A -85,B 0,C 180,E1 4495.653,E2 4495.653} C_VEL
LIN {X 0,Y 189.676,Z 1166.783,A -85,B 0,C 180,E1 4492.316,E2 4492.316} C_VEL
LIN {X 0,Y 171.205,Z 1174.609,A -85,B 0,C 180,E1 4488.205,E2 4488.205} C_VEL
LIN {X 0,Y 151.16,Z 1182.263,A -85,B 0,C 180,E1 4482.268,E2 4482.268} C_VEL
LIN {X 0,Y 130.691,Z 1189.084,A -85,B 0,C 180,E1 4473.523,E2 4473.523} C_VEL
LIN {X 0,Y 116.492,Z 1193.333,A -85,B 0,C 180,E1 4464.291,E2 4464.291} C_VEL
LIN {X 0,Y 106.375,Z 1196.167,A -85,B 0,C 180,E1 4454.071,E2 4454.071} C_VEL
LIN {X 0,Y 99.779,Z 1197.954,A -85,B 0,C 180,E1 4442.672,E2 4442.672} C_VEL
LIN {X 0,Y 96.668,Z 1198.765,A -85,B 0,C 180,E1 4431.224,E2 4431.224} C_VEL
LIN {X 0,Y 95.947,Z 1198.831,A -85,B 0,C 180,E1 4421.42,E2 4421.42} C_VEL
LIN {X 0,Y 95.929,Z 1198.496,A -85,B 0,C 180,E1 4412.987,E2 4412.987} C_VEL
LIN {X 0,Y 96.586,Z 1197.359,A -85,B 0,C 180,E1 4402.864,E2 4402.864} C_VEL
LIN {X 0,Y 100.817,Z 1194.633,A -85,B 0,C 180,E1 4388.473,E2 4388.473} C_VEL
LIN {X 0,Y 109.602,Z 1190.42,A -85,B 0,C 180,E1 4375.556,E2 4375.556} C_VEL
LIN {X 0,Y 120.692,Z 1185.565,A -85,B 0,C 180,E1 4365.902,E2 4365.902} C_VEL
LIN {X 0,Y 133.653,Z 1179.863,A -85,B 0,C 180,E1 4358.233,E2 4358.233} C_VEL
LIN {X 0,Y 149.131,Z 1172.727,A -85,B 0,C 180,E1 4351.627,E2 4351.627} C_VEL
LIN {X 0,Y 169.322,Z 1162.734,A -85,B 0,C 180,E1 4345.382,E2 4345.382} C_VEL
LIN {X 0,Y 190.119,Z 1151.134,A -85,B 0,C 180,E1 4340.59,E2 4340.59} C_VEL
LIN {X 0,Y 207.503,Z 1140.557,A -85,B 0,C 180,E1 4337.434,E2 4337.434} C_VEL
LIN {X 0,Y 224.489,Z 1129.289,A -85,B 0,C 180,E1 4334.873,E2 4334.873} C_VEL
LIN {X 0,Y 243.69,Z 1115.341,A -85,B 0,C 180,E1 4332.443,E2 4332.443} C_VEL
LIN {X 0,Y 265.129,Z 1097.889,A -85,B 0,C 180,E1 4330.172,E2 4330.172} C_VEL
LIN {X 0,Y 282.154,Z 1082.477,A -85,B 0,C 180,E1 4328.63,E2 4328.63} C_VEL
LIN {X 0,Y 297.913,Z 1066.829,A -85,B 0,C 180,E1 4327.363,E2 4327.363} C_VEL
LIN {X 0,Y 313.843,Z 1049.443,A -85,B 0,C 180,E1 4326.219,E2 4326.219} C_VEL
LIN {X 0,Y 333.21,Z 1025.624,A -85,B 0,C 180,E1 4324.981,E2 4324.981} C_VEL
LIN {X 0,Y 346.88,Z 1006.615,A -85,B 0,C 180,E1 4324.198,E2 4324.198} C_VEL
LIN {X 0,Y 357.852,Z 989.757,A -85,B 0,C 180,E1 4323.601,E2 4323.601} C_VEL
LIN {X 0,Y 361.184,Z 990.879,A -85,B 0,C 180,E1 4323.361,E2 4323.361} C_VEL
LIN {X 0,Y 361.184,Z 1038.688,A -85,B 0,C 180,E1 4323.361,E2 4323.361} C_VEL
LIN {X 0,Y 337.686,Z 1038.688,A -85,B 0,C 180,E1 4323.769,E2 4323.769} C_VEL
LIN {X 0,Y 335.698,Z 1036.688,A -85,B 0,C 180,E1 4323.806,E2 4323.806} C_VEL
LIN {X 0,Y 335.698,Z 1028.032,A -85,B 0,C 180,E1 4323.806,E2 4323.806} C_VEL
LIN {X 0,Y 332.286,Z 1026.799,A -85,B 0,C 180,E1 4323.623,E2 4323.623} C_VEL
LIN {X 0,Y 313.259,Z 1049.962,A -85,B 0,C 180,E1 4322.529,E2 4322.529} C_VEL
LIN {X 0,Y 297.878,Z 1066.672,A -85,B 0,C 180,E1 4321.539,E2 4321.539} C_VEL
LIN {X 0,Y 281.966,Z 1082.41,A -85,B 0,C 180,E1 4320.399,E2 4320.399} C_VEL
LIN {X 0,Y 265,Z 1097.703,A -85,B 0,C 180,E1 4319.015,E2 4319.015} C_VEL
LIN {X 0,Y 243.247,Z 1115.38,A -85,B 0,C 180,E1 4316.937,E2 4316.937} C_VEL
LIN {X 0,Y 222.815,Z 1130.087,A -85,B 0,C 180,E1 4314.593,E2 4314.593} C_VEL
LIN {X 0,Y 204.908,Z 1141.815,A -85,B 0,C 180,E1 4312.114,E2 4312.114} C_VEL
LIN {X 0,Y 186.398,Z 1152.877,A -85,B 0,C 180,E1 4309,E2 4309} C_VEL
LIN {X 0,Y 163.325,Z 1165.314,A -85,B 0,C 180,E1 4303.974,E2 4303.974} C_VEL
LIN {X 0,Y 144.172,Z 1174.505,A -85,B 0,C 180,E1 4298.327,E2 4298.327} C_VEL
LIN {X 0,Y 128.137,Z 1181.633,A -85,B 0,C 180,E1 4291.853,E2 4291.853} C_VEL
LIN {X 0,Y 113.987,Z 1187.588,A -85,B 0,C 180,E1 4283.803,E2 4283.803} C_VEL
LIN {X 0,Y 100.345,Z 1193.329,A -85,B 0,C 180,E1 4271.639,E2 4271.639} C_VEL
LIN {X 0,Y 91.206,Z 1197.511,A -85,B 0,C 180,E1 4255.977,E2 4255.977} C_VEL
LIN {X 0,Y 88.316,Z 1199.557,A -85,B 0,C 180,E1 4243.087,E2 4243.087} C_VEL
LIN {X 0,Y 87.915,Z 1200.563,A -85,B 0,C 180,E1 4232.607,E2 4232.607} C_VEL
LIN {X 0,Y 87.937,Z 1200.847,A -85,B 0,C 180,E1 4224.126,E2 4224.126} C_VEL
LIN {X 0,Y 88.865,Z 1200.651,A -85,B 0,C 180,E1 4212.99,E2 4212.99} C_VEL
LIN {X 0,Y 92.559,Z 1199.69,A -85,B 0,C 180,E1 4200.915,E2 4200.915} C_VEL
LIN {X 0,Y 100.247,Z 1197.7,A -85,B 0,C 180,E1 4188.831,E2 4188.831} C_VEL
LIN {X 0,Y 112.484,Z 1194.408,A -85,B 0,C 180,E1 4177.711,E2 4177.711} C_VEL
LIN {X 0,Y 132.245,Z 1188.563,A -85,B 0,C 180,E1 4166.854,E2 4166.854} C_VEL
LIN {X 0,Y 151.992,Z 1181.842,A -85,B 0,C 180,E1 4159.83,E2 4159.83} C_VEL
LIN {X 0,Y 170.789,Z 1174.709,A -85,B 0,C 180,E1 4154.992,E2 4154.992} C_VEL
LIN {X 0,Y 190.538,Z 1166.349,A -85,B 0,C 180,E1 4151.1,E2 4151.1} C_VEL
LIN {X 0,Y 215.721,Z 1154.303,A -85,B 0,C 180,E1 4147.306,E2 4147.306} C_VEL
LIN {X 0,Y 237.768,Z 1142.211,A -85,B 0,C 180,E1 4144.708,E2 4144.708} C_VEL
LIN {X 0,Y 252.749,Z 1133.232,A -85,B 0,C 180,E1 4143.222,E2 4143.222} C_VEL
LIN {X 0,Y 226.903,Z 1148.155,A -85,B 0,C 180,E1 4140.505,E2 4140.505} C_VEL
LIN {X 0,Y 206.126,Z 1158.693,A -85,B 0,C 180,E1 4137.769,E2 4137.769} C_VEL
LIN {X 0,Y 186.8,Z 1167.486,A -85,B 0,C 180,E1 4134.607,E2 4134.607} C_VEL
LIN {X 0,Y 166.218,Z 1175.858,A -85,B 0,C 180,E1 4130.303,E2 4130.303} C_VEL
LIN {X 0,Y 141.919,Z 1184.443,A -85,B 0,C 180,E1 4123.21,E2 4123.21} C_VEL
LIN {X 0,Y 124.626,Z 1189.746,A -85,B 0,C 180,E1 4115.846,E2 4115.846} C_VEL
LIN {X 0,Y 110.667,Z 1193.597,A -85,B 0,C 180,E1 4107.165,E2 4107.165} C_VEL
LIN {X 0,Y 99.459,Z 1196.425,A -85,B 0,C 180,E1 4096.37,E2 4096.37} C_VEL
LIN {X 0,Y 91.958,Z 1198.202,A -85,B 0,C 180,E1 4083.678,E2 4083.678} C_VEL
LIN {X 0,Y 88.528,Z 1198.931,A -85,B 0,C 180,E1 4070.371,E2 4070.371} C_VEL
LIN {X 0,Y 87.934,Z 1198.859,A -85,B 0,C 180,E1 4060.482,E2 4060.482} C_VEL
LIN {X 0,Y 87.944,Z 1198.489,A -85,B 0,C 180,E1 4051.955,E2 4051.955} C_VEL
LIN {X 0,Y 88.952,Z 1197.282,A -85,B 0,C 180,E1 4040.293,E2 4040.293} C_VEL
LIN {X 0,Y 94.287,Z 1194.334,A -85,B 0,C 180,E1 4024.902,E2 4024.902} C_VEL
LIN {X 0,Y 103.513,Z 1190.411,A -85,B 0,C 180,E1 4012.517,E2 4012.517} C_VEL
LIN {X 0,Y 115.614,Z 1185.535,A -85,B 0,C 180,E1 4002.685,E2 4002.685} C_VEL
LIN {X 0,Y 130.192,Z 1179.515,A -85,B 0,C 180,E1 3994.741,E2 3994.741} C_VEL
LIN {X 0,Y 149.05,Z 1171.222,A -85,B 0,C 180,E1 3987.573,E2 3987.573} C_VEL
LIN {X 0,Y 171.03,Z 1160.366,A -85,B 0,C 180,E1 3981.639,E2 3981.639} C_VEL
LIN {X 0,Y 189.169,Z 1150.479,A -85,B 0,C 180,E1 3977.938,E2 3977.938} C_VEL
LIN {X 0,Y 207.02,Z 1139.815,A -85,B 0,C 180,E1 3974.995,E2 3974.995} C_VEL
LIN {X 0,Y 228.086,Z 1125.964,A -85,B 0,C 180,E1 3972.161,E2 3972.161} C_VEL
LIN {X 0,Y 249.595,Z 1109.972,A -85,B 0,C 180,E1 3969.785,E2 3969.785} C_VEL
LIN {X 0,Y 267.634,Z 1095.083,A -85,B 0,C 180,E1 3968.105,E2 3968.105} C_VEL
LIN {X 0,Y 283.944,Z 1080.301,A -85,B 0,C 180,E1 3966.78,E2 3966.78} C_VEL
LIN {X 0,Y 301.359,Z 1062.942,A -85,B 0,C 180,E1 3965.53,E2 3965.53} C_VEL
LIN {X 0,Y 320.363,Z 1041.608,A -85,B 0,C 180,E1 3964.319,E2 3964.319} C_VEL
LIN {X 0,Y 332.286,Z 1026.799,A -85,B 0,C 180,E1 3963.623,E2 3963.623} C_VEL
LIN {X 0,Y 335.626,Z 1028.049,A -85,B 0,C 180,E1 3963.411,E2 3963.411} C_VEL
LIN {X 0,Y 335.626,Z 1068.893,A -85,B 0,C 180,E1 3963.411,E2 3963.411} C_VEL
LIN {X 0,Y 311.431,Z 1068.893,A -85,B 0,C 180,E1 3963.907,E2 3963.907} C_VEL
LIN {X 0,Y 309.445,Z 1066.893,A -85,B 0,C 180,E1 3963.951,E2 3963.951} C_VEL
LIN {X 0,Y 309.445,Z 1058.845,A -85,B 0,C 180,E1 3963.951,E2 3963.951} C_VEL
LIN {X 0,Y 306.455,Z 1057.417,A -85,B 0,C 180,E1 3963.65,E2 3963.65} C_VEL
LIN {X 0,Y 285.698,Z 1078.532,A -85,B 0,C 180,E1 3962.346,E2 3962.346} C_VEL
LIN {X 0,Y 268.031,Z 1094.566,A -85,B 0,C 180,E1 3961.069,E2 3961.069} C_VEL
LIN {X 0,Y 251.966,Z 1107.865,A -85,B 0,C 180,E1 3959.743,E2 3959.743} C_VEL
LIN {X 0,Y 234.101,Z 1121.365,A -85,B 0,C 180,E1 3958.051,E2 3958.051} C_VEL
LIN {X 0,Y 211.628,Z 1136.723,A -85,B 0,C 180,E1 3955.478,E2 3955.478} C_VEL
LIN {X 0,Y 189.664,Z 1149.883,A -85,B 0,C 180,E1 3952.342,E2 3952.342} C_VEL
LIN {X 0,Y 171.116,Z 1159.951,A -85,B 0,C 180,E1 3949.006,E2 3949.006} C_VEL
LIN {X 0,Y 152.871,Z 1168.953,A -85,B 0,C 180,E1 3944.833,E2 3944.833} C_VEL
LIN {X 0,Y 131.41,Z 1178.601,A -85,B 0,C 180,E1 3938.109,E2 3938.109} C_VEL
LIN {X 0,Y 111.967,Z 1186.326,A -85,B 0,C 180,E1 3929.011,E2 3929.011} C_VEL
LIN {X 0,Y 98.723,Z 1191.37,A -85,B 0,C 180,E1 3919.428,E2 3919.428} C_VEL
LIN {X 0,Y 88.897,Z 1195.179,A -85,B 0,C 180,E1 3908.062,E2 3908.062} C_VEL
LIN {X 0,Y 82.623,Z 1197.985,A -85,B 0,C 180,E1 3894.819,E2 3894.819} C_VEL
LIN {X 0,Y 80.224,Z 1199.646,A -85,B 0,C 180,E1 3882.232,E2 3882.232} C_VEL
LIN {X 0,Y 79.916,Z 1200.488,A -85,B 0,C 180,E1 3872.151,E2 3872.151} C_VEL
LIN {X 0,Y 79.967,Z 1200.769,A -85,B 0,C 180,E1 3862.817,E2 3862.817} C_VEL
LIN {X 0,Y 81.576,Z 1200.497,A -85,B 0,C 180,E1 3849.179,E2 3849.179} C_VEL
LIN {X 0,Y 89.127,Z 1198.924,A -85,B 0,C 180,E1 3831.902,E2 3831.902} C_VEL
LIN {X 0,Y 103.129,Z 1195.518,A -85,B 0,C 180,E1 3817.344,E2 3817.344} C_VEL
LIN {X 0,Y 118.752,Z 1191.389,A -85,B 0,C 180,E1 3807.863,E2 3807.863} C_VEL
LIN {X 0,Y 135.909,Z 1186.311,A -85,B 0,C 180,E1 3800.882,E2 3800.882} C_VEL
LIN {X 0,Y 156.311,Z 1179.491,A -85,B 0,C 180,E1 3795.009,E2 3795.009} C_VEL
LIN {X 0,Y 182.576,Z 1169.265,A -85,B 0,C 180,E1 3789.684,E2 3789.684} C_VEL
LIN {X 0,Y 203.299,Z 1160.004,A -85,B 0,C 180,E1 3786.554,E2 3786.554} C_VEL
LIN {X 0,Y 222.57,Z 1150.4,A -85,B 0,C 180,E1 3784.214,E2 3784.214} C_VEL
LIN {X 0,Y 232.069,Z 1145.38,A -85,B 0,C 180,E1 3783.211,E2 3783.211} C_VEL
LIN {X 0,Y 207.977,Z 1157.609,A -85,B 0,C 180,E1 3780.457,E2 3780.457} C_VEL
LIN {X 0,Y 187.159,Z 1166.953,A -85,B 0,C 180,E1 3777.448,E2 3777.448} C_VEL
LIN {X 0,Y 167.479,Z 1174.808,A -85,B 0,C 180,E1 3773.831,E2 3773.831} C_VEL
LIN {X 0,Y 145.835,Z 1182.448,A -85,B 0,C 180,E1 3768.531,E2 3768.531} C_VEL
LIN {X 0,Y 123.105,Z 1189.256,A -85,B 0,C 180,E1 3760.416,E2 3760.416} C_VEL
LIN {X 0,Y 106.754,Z 1193.477,A -85,B 0,C 180,E1 3751.466,E2 3751.466} C_VEL
LIN {X 0,Y 94.249,Z 1196.345,A -85,B 0,C 180,E1 3740.754,E2 3740.754} C_VEL
LIN {X 0,Y 85.339,Z 1198.192,A -85,B 0,C 180,E1 3727.535,E2 3727.535} C_VEL
LIN {X 0,Y 81.036,Z 1198.965,A -85,B 0,C 180,E1 3714.027,E2 3714.027} C_VEL
LIN {X 0,Y 79.974,Z 1199.001,A -85,B 0,C 180,E1 3702.783,E2 3702.783} C_VEL
LIN {X 0,Y 79.923,Z 1198.701,A -85,B 0,C 180,E1 3693.586,E2 3693.586} C_VEL
LIN {X 0,Y 80.622,Z 1197.67,A -85,B 0,C 180,E1 3682.159,E2 3682.159} C_VEL
LIN {X 0,Y 85.417,Z 1195.23,A -85,B 0,C 180,E1 3665.814,E2 3665.814} C_VEL
LIN {X 0,Y 96.696,Z 1190.807,A -85,B 0,C 180,E1 3650.127,E2 3650.127} C_VEL
LIN {X 0,Y 109.624,Z 1186.002,A -85,B 0,C 180,E1 3639.991,E2 3639.991} C_VEL
LIN {X 0,Y 124.994,Z 1180.055,A -85,B 0,C 180,E1 3632.014,E2 3632.014} C_VEL
LIN {X 0,Y 142.088,Z 1172.922,A -85,B 0,C 180,E1 3625.747,E2 3625.747} C_VEL
LIN {X 0,Y 164.183,Z 1162.771,A -85,B 0,C 180,E1 3619.941,E2 3619.941} C_VEL
LIN {X 0,Y 185.924,Z 1151.331,A -85,B 0,C 180,E1 3615.716,E2 3615.716} C_VEL
LIN {X 0,Y 204.146,Z 1140.75,A -85,B 0,C 180,E1 3612.929,E2 3612.929} C_VEL
LIN {X 0,Y 222.754,Z 1128.855,A -85,B 0,C 180,E1 3610.579,E2 3610.579} C_VEL
LIN {X 0,Y 244.529,Z 1113.456,A -85,B 0,C 180,E1 3608.305,E2 3608.305} C_VEL
LIN {X 0,Y 265.65,Z 1096.418,A -85,B 0,C 180,E1 3606.464,E2 3606.464} C_VEL
LIN {X 0,Y 282.133,Z 1081.753,A -85,B 0,C 180,E1 3605.229,E2 3605.229} C_VEL
LIN {X 0,Y 297.751,Z 1066.511,A -85,B 0,C 180,E1 3604.187,E2 3604.187} C_VEL
LIN {X 0,Y 306.455,Z 1057.417,A -85,B 0,C 180,E1 3603.65,E2 3603.65} C_VEL
LIN {X 0,Y 300.467,Z 1063.908,A -85,B 0,C 180,E1 3603.251,E2 3603.251} C_VEL
LIN {X 0,Y 293.035,Z 1071.521,A -85,B 0,C 180,E1 3603.175,E2 3603.175} C_VEL
LIN {X 0,Y 283.071,Z 1081.066,A -85,B 0,C 180,E1 3603.531,E2 3603.531} C_VEL
LIN {X 0,Y 271.689,Z 1091.139,A -85,B 0,C 180,E1 3604.25,E2 3604.25} C_VEL
LIN {X 0,Y 253.181,Z 1106.381,A -85,B 0,C 180,E1 3605.621,E2 3605.621} C_VEL
LIN {X 0,Y 235.779,Z 1119.394,A -85,B 0,C 180,E1 3607.11,E2 3607.11} C_VEL
LIN {X 0,Y 217.602,Z 1131.745,A -85,B 0,C 180,E1 3608.923,E2 3608.923} C_VEL
LIN {X 0,Y 195.007,Z 1145.611,A -85,B 0,C 180,E1 3611.676,E2 3611.676} C_VEL
LIN {X 0,Y 172.027,Z 1157.865,A -85,B 0,C 180,E1 3615.242,E2 3615.242} C_VEL
LIN {X 0,Y 153.023,Z 1166.959,A -85,B 0,C 180,E1 3619.07,E2 3619.07} C_VEL
LIN {X 0,Y 135.403,Z 1174.572,A -85,B 0,C 180,E1 3623.701,E2 3623.701} C_VEL
LIN {X 0,Y 116.258,Z 1182.076,A -85,B 0,C 180,E1 3630.68,E2 3630.68} C_VEL
LIN {X 0,Y 96.008,Z 1189.185,A -85,B 0,C 180,E1 3642.318,E2 3642.318} C_VEL
LIN {X 0,Y 83.882,Z 1193.268,A -85,B 0,C 180,E1 3654.263,E2 3654.263} C_VEL
LIN {X 0,Y 75.965,Z 1196.152,A -85,B 0,C 180,E1 3668.375,E2 3668.375} C_VEL
LIN {X 0,Y 72.502,Z 1197.926,A -85,B 0,C 180,E1 3682.87,E2 3682.87} C_VEL
LIN {X 0,Y 71.919,Z 1198.823,A -85,B 0,C 180,E1 3694.785,E2 3694.785} C_VEL
LIN {X 0,Y 72.068,Z 1199.135,A -85,B 0,C 180,E1 3705.284,E2 3705.284} C_VEL
LIN {X 0,Y 74.469,Z 1198.943,A -85,B 0,C 180,E1 3720.677,E2 3720.677} C_VEL
LIN {X 0,Y 83.614,Z 1197.504,A -85,B 0,C 180,E1 3738.882,E2 3738.882} C_VEL
LIN {X 0,Y 99.431,Z 1194.252,A -85,B 0,C 180,E1 3753.504,E2 3753.504} C_VEL
LIN {X 0,Y 115.86,Z 1190.39,A -85,B 0,C 180,E1 3762.419,E2 3762.419} C_VEL
LIN {X 0,Y 134.379,Z 1185.358,A -85,B 0,C 180,E1 3769.159,E2 3769.159} C_VEL
LIN {X 0,Y 157.573,Z 1178.063,A -85,B 0,C 180,E1 3775.014,E2 3775.014} C_VEL
LIN {X 0,Y 182.979,Z 1168.479,A -85,B 0,C 180,E1 3779.538,E2 3779.538} C_VEL
LIN {X 0,Y 203.129,Z 1159.795,A -85,B 0,C 180,E1 3782.263,E2 3782.263} C_VEL
LIN {X 0,Y 211.083,Z 1156.158,A -85,B 0,C 180,E1 3783.215,E2 3783.215} C_VEL
LIN {X 0,Y 187.843,Z 1166.647,A -85,B 0,C 180,E1 3786.111,E2 3786.111} C_VEL
LIN {X 0,Y 167.234,Z 1174.878,A -85,B 0,C 180,E1 3789.426,E2 3789.426} C_VEL
LIN {X 0,Y 146.256,Z 1182.261,A -85,B 0,C 180,E1 3793.89,E2 3793.89} C_VEL
LIN {X 0,Y 121.462,Z 1189.745,A -85,B 0,C 180,E1 3801.534,E2 3801.534} C_VEL
LIN {X 0,Y 102.412,Z 1194.539,A -85,B 0,C 180,E1 3810.779,E2 3810.779} C_VEL
LIN {X 0,Y 88.427,Z 1197.627,A -85,B 0,C 180,E1 3821.731,E2 3821.731} C_VEL
LIN {X 0,Y 78.582,Z 1199.574,A -85,B 0,C 180,E1 3835.07,E2 3835.07} C_VEL
LIN {X 0,Y 73.443,Z 1200.494,A -85,B 0,C 180,E1 3849.27,E2 3849.27} C_VEL
